   1:L PR[91] 10mm/sec CNT100;
   1:  PR[GP1:91,1] = PR[GP1:90,1] + -17.777;
   1:  PR[GP1:91,2] = PR[GP1:90,2] + -17.049;
   1:L PR[91] 10mm/sec CNT100;
   1:  PR[GP1:91,1] = PR[GP1:90,1] + -17.068;
   1:  PR[GP1:91,2] = PR[GP1:90,2] + -16.935;
   1:L PR[91] 10mm/sec CNT100;
   1:  PR[GP1:91,1] = PR[GP1:90,1] + -14.386;
   1:  PR[GP1:91,2] = PR[GP1:90,2] + -16.296;
   1:L PR[91] 10mm/sec CNT100;
   1:  PR[GP1:91,1] = PR[GP1:90,1] + -13.899;
   1:  PR[GP1:91,2] = PR[GP1:90,2] + -16.133;
   1:L PR[91] 10mm/sec CNT100;
   1:  PR[GP1:91,1] = PR[GP1:90,1] + -11.116;
   1:  PR[GP1:91,2] = PR[GP1:90,2] + -14.804;
   1:L PR[91] 10mm/sec CNT100;
   1:  PR[GP1:91,1] = PR[GP1:90,1] + -10.848;
   1:  PR[GP1:91,2] = PR[GP1:90,2] + -14.661;
   1:L PR[91] 10mm/sec CNT100;
   1:  PR[GP1:91,1] = PR[GP1:90,1] + -8.058;
   1:  PR[GP1:91,2] = PR[GP1:90,2] + -12.514;
   1:L PR[91] 10mm/sec CNT100;
   1:  PR[GP1:91,1] = PR[GP1:90,1] + -7.983;
   1:  PR[GP1:91,2] = PR[GP1:90,2] + -12.434;
   1:L PR[91] 10mm/sec CNT100;
   1:  PR[GP1:91,1] = PR[GP1:90,1] + -5.754;
   1:  PR[GP1:91,2] = PR[GP1:90,2] + -9.796;
   1:L PR[91] 10mm/sec CNT100;
   1:  PR[GP1:91,1] = PR[GP1:90,1] + -4.074;
   1:  PR[GP1:91,2] = PR[GP1:90,2] + -6.675;
   1:L PR[91] 10mm/sec CNT100;
   1:  PR[GP1:91,1] = PR[GP1:90,1] + -3.054;
   1:  PR[GP1:91,2] = PR[GP1:90,2] + -3.139;
   1:L PR[91] 10mm/sec CNT100;
   1:  PR[GP1:91,1] = PR[GP1:90,1] + -2.957;
   1:  PR[GP1:91,2] = PR[GP1:90,2] + -2.843;
   1:L PR[91] 10mm/sec CNT100;
   1:  PR[GP1:91,1] = PR[GP1:90,1] + -2.891;
   1:  PR[GP1:91,2] = PR[GP1:90,2] + -2.753;
   1:L PR[91] 10mm/sec CNT100;
   1:  PR[GP1:91,1] = PR[GP1:90,1] + -2.846;
   1:  PR[GP1:91,2] = PR[GP1:90,2] + -2.649;
   1:L PR[91] 10mm/sec CNT100;
   1:  PR[GP1:91,1] = PR[GP1:90,1] + -2.751;
   1:  PR[GP1:91,2] = PR[GP1:90,2] + -2.377;
   1:L PR[91] 10mm/sec CNT100;
   1:  PR[GP1:91,1] = PR[GP1:90,1] + -2.564;
   1:  PR[GP1:91,2] = PR[GP1:90,2] + -2.018;
   1:L PR[91] 10mm/sec CNT100;
   1:  PR[GP1:91,1] = PR[GP1:90,1] + -2.286;
   1:  PR[GP1:91,2] = PR[GP1:90,2] + -1.644;
   1:L PR[91] 10mm/sec CNT100;
   1:  PR[GP1:91,1] = PR[GP1:90,1] + -1.981;
   1:  PR[GP1:91,2] = PR[GP1:90,2] + -1.337;
   1:L PR[91] 10mm/sec CNT100;
   1:  PR[GP1:91,1] = PR[GP1:90,1] + -1.497;
   1:  PR[GP1:91,2] = PR[GP1:90,2] + -1.028;
   1:L PR[91] 10mm/sec CNT100;
   1:  PR[GP1:91,1] = PR[GP1:90,1] + -1.290;
   1:  PR[GP1:91,2] = PR[GP1:90,2] + -0.917;
   1:L PR[91] 10mm/sec CNT100;
   1:  PR[GP1:91,1] = PR[GP1:90,1] + -0.204;
   1:  PR[GP1:91,2] = PR[GP1:90,2] + -0.687;
   1:L PR[91] 10mm/sec CNT100;
   1:  PR[GP1:91,1] = PR[GP1:90,1] + 0.891;
   1:  PR[GP1:91,2] = PR[GP1:90,2] + -0.965;
   1:L PR[91] 10mm/sec CNT100;
   1:  PR[GP1:91,1] = PR[GP1:90,1] + 1.190;
   1:  PR[GP1:91,2] = PR[GP1:90,2] + -1.125;
   1:L PR[91] 10mm/sec CNT100;
   1:  PR[GP1:91,1] = PR[GP1:90,1] + 1.414;
   1:  PR[GP1:91,2] = PR[GP1:90,2] + -1.278;
   1:L PR[91] 10mm/sec CNT100;
   1:  PR[GP1:91,1] = PR[GP1:90,1] + 2.090;
   1:  PR[GP1:91,2] = PR[GP1:90,2] + -1.951;
   1:L PR[91] 10mm/sec CNT100;
   1:  PR[GP1:91,1] = PR[GP1:90,1] + 2.234;
   1:  PR[GP1:91,2] = PR[GP1:90,2] + -2.141;
   1:L PR[91] 10mm/sec CNT100;
   1:  PR[GP1:91,1] = PR[GP1:90,1] + 2.617;
   1:  PR[GP1:91,2] = PR[GP1:90,2] + -3.082;
   1:L PR[91] 10mm/sec CNT100;
   1:  PR[GP1:91,1] = PR[GP1:90,1] + 3.318;
   1:  PR[GP1:91,2] = PR[GP1:90,2] + -5.804;
   1:L PR[91] 10mm/sec CNT100;
   1:  PR[GP1:91,1] = PR[GP1:90,1] + 4.418;
   1:  PR[GP1:91,2] = PR[GP1:90,2] + -8.231;
   1:L PR[91] 10mm/sec CNT100;
   1:  PR[GP1:91,1] = PR[GP1:90,1] + 5.923;
   1:  PR[GP1:91,2] = PR[GP1:90,2] + -10.467;
   1:L PR[91] 10mm/sec CNT100;
   1:  PR[GP1:91,1] = PR[GP1:90,1] + 7.757;
   1:  PR[GP1:91,2] = PR[GP1:90,2] + -12.452;
   1:L PR[91] 10mm/sec CNT100;
   1:  PR[GP1:91,1] = PR[GP1:90,1] + 9.893;
   1:  PR[GP1:91,2] = PR[GP1:90,2] + -14.128;
   1:L PR[91] 10mm/sec CNT100;
   1:  PR[GP1:91,1] = PR[GP1:90,1] + 12.262;
   1:  PR[GP1:91,2] = PR[GP1:90,2] + -15.460;
   1:L PR[91] 10mm/sec CNT100;
   1:  PR[GP1:91,1] = PR[GP1:90,1] + 14.756;
   1:  PR[GP1:91,2] = PR[GP1:90,2] + -16.425;
   1:L PR[91] 10mm/sec CNT100;
   1:  PR[GP1:91,1] = PR[GP1:90,1] + 17.367;
   1:  PR[GP1:91,2] = PR[GP1:90,2] + -16.996;
   1:L PR[91] 10mm/sec CNT100;
   1:  PR[GP1:91,1] = PR[GP1:90,1] + 20.036;
   1:  PR[GP1:91,2] = PR[GP1:90,2] + -17.161;
   1:L PR[91] 10mm/sec CNT100;
   1:  PR[GP1:91,1] = PR[GP1:90,1] + 22.699;
   1:  PR[GP1:91,2] = PR[GP1:90,2] + -16.917;
   1:L PR[91] 10mm/sec CNT100;
   1:  PR[GP1:91,1] = PR[GP1:90,1] + 25.303;
   1:  PR[GP1:91,2] = PR[GP1:90,2] + -16.264;
   1:L PR[91] 10mm/sec CNT100;
   1:  PR[GP1:91,1] = PR[GP1:90,1] + 27.687;
   1:  PR[GP1:91,2] = PR[GP1:90,2] + -15.253;
   1:L PR[91] 10mm/sec CNT100;
   1:  PR[GP1:91,1] = PR[GP1:90,1] + 29.800;
   1:  PR[GP1:91,2] = PR[GP1:90,2] + -13.948;
   1:L PR[91] 10mm/sec CNT100;
   1:  PR[GP1:91,1] = PR[GP1:90,1] + 30.069;
   1:  PR[GP1:91,2] = PR[GP1:90,2] + -13.749;
   1:L PR[91] 10mm/sec CNT100;
   1:  PR[GP1:91,1] = PR[GP1:90,1] + 31.620;
   1:  PR[GP1:91,2] = PR[GP1:90,2] + -12.411;
   1:L PR[91] 10mm/sec CNT100;
   1:  PR[GP1:91,1] = PR[GP1:90,1] + 31.946;
   1:  PR[GP1:91,2] = PR[GP1:90,2] + -12.109;
   1:L PR[91] 10mm/sec CNT100;
   1:  PR[GP1:91,1] = PR[GP1:90,1] + 33.516;
   1:  PR[GP1:91,2] = PR[GP1:90,2] + -10.262;
   1:L PR[91] 10mm/sec CNT100;
   1:  PR[GP1:91,1] = PR[GP1:90,1] + 33.815;
   1:  PR[GP1:91,2] = PR[GP1:90,2] + -9.828;
   1:L PR[91] 10mm/sec CNT100;
   1:  PR[GP1:91,1] = PR[GP1:90,1] + 34.762;
   1:  PR[GP1:91,2] = PR[GP1:90,2] + -8.269;
   1:L PR[91] 10mm/sec CNT100;
   1:  PR[GP1:91,1] = PR[GP1:90,1] + 35.043;
   1:  PR[GP1:91,2] = PR[GP1:90,2] + -7.748;
   1:L PR[91] 10mm/sec CNT100;
   1:  PR[GP1:91,1] = PR[GP1:90,1] + 35.944;
   1:  PR[GP1:91,2] = PR[GP1:90,2] + -5.545;
   1:L PR[91] 10mm/sec CNT100;
   1:  PR[GP1:91,1] = PR[GP1:90,1] + 36.117;
   1:  PR[GP1:91,2] = PR[GP1:90,2] + -4.929;
   1:L PR[91] 10mm/sec CNT100;
   1:  PR[GP1:91,1] = PR[GP1:90,1] + 36.509;
   1:  PR[GP1:91,2] = PR[GP1:90,2] + -3.281;
   1:L PR[91] 10mm/sec CNT100;
   1:  PR[GP1:91,1] = PR[GP1:90,1] + 36.618;
   1:  PR[GP1:91,2] = PR[GP1:90,2] + -2.625;
   1:L PR[91] 10mm/sec CNT100;
   1:  PR[GP1:91,1] = PR[GP1:90,1] + 36.657;
   1:  PR[GP1:91,2] = PR[GP1:90,2] + -1.925;
   1:L PR[91] 10mm/sec CNT100;
   1:  PR[GP1:91,1] = PR[GP1:90,1] + 36.816;
   1:  PR[GP1:91,2] = PR[GP1:90,2] + -0.277;
   1:L PR[91] 10mm/sec CNT100;
   1:  PR[GP1:91,1] = PR[GP1:90,1] + 36.466;
   1:  PR[GP1:91,2] = PR[GP1:90,2] + 3.030;
   1:L PR[91] 10mm/sec CNT100;
   1:  PR[GP1:91,1] = PR[GP1:90,1] + 35.808;
   1:  PR[GP1:91,2] = PR[GP1:90,2] + 5.173;
   1:L PR[91] 10mm/sec CNT100;
   1:  PR[GP1:91,1] = PR[GP1:90,1] + 35.611;
   1:  PR[GP1:91,2] = PR[GP1:90,2] + 5.902;
   1:L PR[91] 10mm/sec CNT100;
   1:  PR[GP1:91,1] = PR[GP1:90,1] + 35.499;
   1:  PR[GP1:91,2] = PR[GP1:90,2] + 6.196;
   1:L PR[91] 10mm/sec CNT100;
   1:  PR[GP1:91,1] = PR[GP1:90,1] + 33.908;
   1:  PR[GP1:91,2] = PR[GP1:90,2] + 9.143;
   1:L PR[91] 10mm/sec CNT100;
   1:  PR[GP1:91,1] = PR[GP1:90,1] + 32.344;
   1:  PR[GP1:91,2] = PR[GP1:90,2] + 11.025;
   1:L PR[91] 10mm/sec CNT100;
   1:  PR[GP1:91,1] = PR[GP1:90,1] + 32.162;
   1:  PR[GP1:91,2] = PR[GP1:90,2] + 11.277;
   1:L PR[91] 10mm/sec CNT100;
   1:  PR[GP1:91,1] = PR[GP1:90,1] + 31.790;
   1:  PR[GP1:91,2] = PR[GP1:90,2] + 11.697;
   1:L PR[91] 10mm/sec CNT100;
   1:  PR[GP1:91,1] = PR[GP1:90,1] + 29.195;
   1:  PR[GP1:91,2] = PR[GP1:90,2] + 13.796;
   1:L PR[91] 10mm/sec CNT100;
   1:  PR[GP1:91,1] = PR[GP1:90,1] + 26.248;
   1:  PR[GP1:91,2] = PR[GP1:90,2] + 15.339;
   1:L PR[91] 10mm/sec CNT100;
   1:  PR[GP1:91,1] = PR[GP1:90,1] + 23.089;
   1:  PR[GP1:91,2] = PR[GP1:90,2] + 16.266;
   1:L PR[91] 10mm/sec CNT100;
   1:  PR[GP1:91,1] = PR[GP1:90,1] + 19.713;
   1:  PR[GP1:91,2] = PR[GP1:90,2] + 16.557;
   1:L PR[91] 10mm/sec CNT100;
   1:  PR[GP1:91,1] = PR[GP1:90,1] + 16.351;
   1:  PR[GP1:91,2] = PR[GP1:90,2] + 16.182;
   1:L PR[91] 10mm/sec CNT100;
   1:  PR[GP1:91,1] = PR[GP1:90,1] + 13.131;
   1:  PR[GP1:91,2] = PR[GP1:90,2] + 15.163;
   1:L PR[91] 10mm/sec CNT100;
   1:  PR[GP1:91,1] = PR[GP1:90,1] + 10.178;
   1:  PR[GP1:91,2] = PR[GP1:90,2] + 13.541;
   1:L PR[91] 10mm/sec CNT100;
   1:  PR[GP1:91,1] = PR[GP1:90,1] + 7.542;
   1:  PR[GP1:91,2] = PR[GP1:90,2] + 11.371;
   1:L PR[91] 10mm/sec CNT100;
   1:  PR[GP1:91,1] = PR[GP1:90,1] + 5.385;
   1:  PR[GP1:91,2] = PR[GP1:90,2] + 8.744;
   1:L PR[91] 10mm/sec CNT100;
   1:  PR[GP1:91,1] = PR[GP1:90,1] + 3.746;
   1:  PR[GP1:91,2] = PR[GP1:90,2] + 5.756;
   1:L PR[91] 10mm/sec CNT100;
   1:  PR[GP1:91,1] = PR[GP1:90,1] + 2.740;
   1:  PR[GP1:91,2] = PR[GP1:90,2] + 2.534;
   1:L PR[91] 10mm/sec CNT100;
   1:  PR[GP1:91,1] = PR[GP1:90,1] + 2.273;
   1:  PR[GP1:91,2] = PR[GP1:90,2] + 1.475;
   1:L PR[91] 10mm/sec CNT100;
   1:  PR[GP1:91,1] = PR[GP1:90,1] + 1.462;
   1:  PR[GP1:91,2] = PR[GP1:90,2] + 0.697;
   1:L PR[91] 10mm/sec CNT100;
   1:  PR[GP1:91,1] = PR[GP1:90,1] + 1.135;
   1:  PR[GP1:91,2] = PR[GP1:90,2] + 0.502;
   1:L PR[91] 10mm/sec CNT100;
   1:  PR[GP1:91,1] = PR[GP1:90,1] + 0.670;
   1:  PR[GP1:91,2] = PR[GP1:90,2] + 0.285;
   1:L PR[91] 10mm/sec CNT100;
   1:  PR[GP1:91,1] = PR[GP1:90,1] + -0.451;
   1:  PR[GP1:91,2] = PR[GP1:90,2] + 0.136;
   1:L PR[91] 10mm/sec CNT100;
   1:  PR[GP1:91,1] = PR[GP1:90,1] + -1.415;
   1:  PR[GP1:91,2] = PR[GP1:90,2] + 0.419;
   1:L PR[91] 10mm/sec CNT100;
   1:  PR[GP1:91,1] = PR[GP1:90,1] + -1.565;
   1:  PR[GP1:91,2] = PR[GP1:90,2] + 0.501;
   1:L PR[91] 10mm/sec CNT100;
   1:  PR[GP1:91,1] = PR[GP1:90,1] + -1.924;
   1:  PR[GP1:91,2] = PR[GP1:90,2] + 0.759;
   1:L PR[91] 10mm/sec CNT100;
   1:  PR[GP1:91,1] = PR[GP1:90,1] + -2.230;
   1:  PR[GP1:91,2] = PR[GP1:90,2] + 1.037;
   1:L PR[91] 10mm/sec CNT100;
   1:  PR[GP1:91,1] = PR[GP1:90,1] + -2.571;
   1:  PR[GP1:91,2] = PR[GP1:90,2] + 1.459;
   1:L PR[91] 10mm/sec CNT100;
   1:  PR[GP1:91,1] = PR[GP1:90,1] + -2.686;
   1:  PR[GP1:91,2] = PR[GP1:90,2] + 1.725;
   1:L PR[91] 10mm/sec CNT100;
   1:  PR[GP1:91,1] = PR[GP1:90,1] + -2.840;
   1:  PR[GP1:91,2] = PR[GP1:90,2] + 2.011;
   1:L PR[91] 10mm/sec CNT100;
   1:  PR[GP1:91,1] = PR[GP1:90,1] + -2.897;
   1:  PR[GP1:91,2] = PR[GP1:90,2] + 2.157;
   1:L PR[91] 10mm/sec CNT100;
   1:  PR[GP1:91,1] = PR[GP1:90,1] + -2.963;
   1:  PR[GP1:91,2] = PR[GP1:90,2] + 2.160;
   1:L PR[91] 10mm/sec CNT100;
   1:  PR[GP1:91,1] = PR[GP1:90,1] + -4.071;
   1:  PR[GP1:91,2] = PR[GP1:90,2] + 6.022;
   1:L PR[91] 10mm/sec CNT100;
   1:  PR[GP1:91,1] = PR[GP1:90,1] + -4.185;
   1:  PR[GP1:91,2] = PR[GP1:90,2] + 6.274;
   1:L PR[91] 10mm/sec CNT100;
   1:  PR[GP1:91,1] = PR[GP1:90,1] + -5.644;
   1:  PR[GP1:91,2] = PR[GP1:90,2] + 8.982;
   1:L PR[91] 10mm/sec CNT100;
   1:  PR[GP1:91,1] = PR[GP1:90,1] + -5.914;
   1:  PR[GP1:91,2] = PR[GP1:90,2] + 9.386;
   1:L PR[91] 10mm/sec CNT100;
   1:  PR[GP1:91,1] = PR[GP1:90,1] + -7.700;
   1:  PR[GP1:91,2] = PR[GP1:90,2] + 11.479;
   1:L PR[91] 10mm/sec CNT100;
   1:  PR[GP1:91,1] = PR[GP1:90,1] + -8.173;
   1:  PR[GP1:91,2] = PR[GP1:90,2] + 11.985;
   1:L PR[91] 10mm/sec CNT100;
   1:  PR[GP1:91,1] = PR[GP1:90,1] + -10.830;
   1:  PR[GP1:91,2] = PR[GP1:90,2] + 14.014;
   1:L PR[91] 10mm/sec CNT100;
   1:  PR[GP1:91,1] = PR[GP1:90,1] + -11.609;
   1:  PR[GP1:91,2] = PR[GP1:90,2] + 14.428;
   1:L PR[91] 10mm/sec CNT100;
   1:  PR[GP1:91,1] = PR[GP1:90,1] + -13.732;
   1:  PR[GP1:91,2] = PR[GP1:90,2] + 15.431;
   1:L PR[91] 10mm/sec CNT100;
   1:  PR[GP1:91,1] = PR[GP1:90,1] + -14.726;
   1:  PR[GP1:91,2] = PR[GP1:90,2] + 15.765;
   1:L PR[91] 10mm/sec CNT100;
   1:  PR[GP1:91,1] = PR[GP1:90,1] + -16.776;
   1:  PR[GP1:91,2] = PR[GP1:90,2] + 16.244;
   1:L PR[91] 10mm/sec CNT100;
   1:  PR[GP1:91,1] = PR[GP1:90,1] + -17.943;
   1:  PR[GP1:91,2] = PR[GP1:90,2] + 16.432;
   1:L PR[91] 10mm/sec CNT100;
   1:  PR[GP1:91,1] = PR[GP1:90,1] + -19.155;
   1:  PR[GP1:91,2] = PR[GP1:90,2] + 16.425;
   1:L PR[91] 10mm/sec CNT100;
   1:  PR[GP1:91,1] = PR[GP1:90,1] + -21.180;
   1:  PR[GP1:91,2] = PR[GP1:90,2] + 16.457;
   1:L PR[91] 10mm/sec CNT100;
   1:  PR[GP1:91,1] = PR[GP1:90,1] + -22.467;
   1:  PR[GP1:91,2] = PR[GP1:90,2] + 16.236;
   1:L PR[91] 10mm/sec CNT100;
   1:  PR[GP1:91,1] = PR[GP1:90,1] + -24.282;
   1:  PR[GP1:91,2] = PR[GP1:90,2] + 15.879;
   1:L PR[91] 10mm/sec CNT100;
   1:  PR[GP1:91,1] = PR[GP1:90,1] + -25.602;
   1:  PR[GP1:91,2] = PR[GP1:90,2] + 15.419;
   1:L PR[91] 10mm/sec CNT100;
   1:  PR[GP1:91,1] = PR[GP1:90,1] + -27.180;
   1:  PR[GP1:91,2] = PR[GP1:90,2] + 14.741;
   1:L PR[91] 10mm/sec CNT100;
   1:  PR[GP1:91,1] = PR[GP1:90,1] + -28.470;
   1:  PR[GP1:91,2] = PR[GP1:90,2] + 14.037;
   1:L PR[91] 10mm/sec CNT100;
   1:  PR[GP1:91,1] = PR[GP1:90,1] + -29.792;
   1:  PR[GP1:91,2] = PR[GP1:90,2] + 13.097;
   1:L PR[91] 10mm/sec CNT100;
   1:  PR[GP1:91,1] = PR[GP1:90,1] + -30.990;
   1:  PR[GP1:91,2] = PR[GP1:90,2] + 12.159;
   1:L PR[91] 10mm/sec CNT100;
   1:  PR[GP1:91,1] = PR[GP1:90,1] + -33.104;
   1:  PR[GP1:91,2] = PR[GP1:90,2] + 9.848;
   1:L PR[91] 10mm/sec CNT100;
   1:  PR[GP1:91,1] = PR[GP1:90,1] + -33.952;
   1:  PR[GP1:91,2] = PR[GP1:90,2] + 8.545;
   1:L PR[91] 10mm/sec CNT100;
   1:  PR[GP1:91,1] = PR[GP1:90,1] + -34.734;
   1:  PR[GP1:91,2] = PR[GP1:90,2] + 7.207;
   1:L PR[91] 10mm/sec CNT100;
   1:  PR[GP1:91,1] = PR[GP1:90,1] + -35.363;
   1:  PR[GP1:91,2] = PR[GP1:90,2] + 5.766;
   1:L PR[91] 10mm/sec CNT100;
   1:  PR[GP1:91,1] = PR[GP1:90,1] + -35.844;
   1:  PR[GP1:91,2] = PR[GP1:90,2] + 4.309;
   1:L PR[91] 10mm/sec CNT100;
   1:  PR[GP1:91,1] = PR[GP1:90,1] + -36.227;
   1:  PR[GP1:91,2] = PR[GP1:90,2] + 2.791;
   1:L PR[91] 10mm/sec CNT100;
   1:  PR[GP1:91,1] = PR[GP1:90,1] + -36.358;
   1:  PR[GP1:91,2] = PR[GP1:90,2] + 1.200;
   1:L PR[91] 10mm/sec CNT100;
   1:  PR[GP1:91,1] = PR[GP1:90,1] + -36.519;
   1:  PR[GP1:91,2] = PR[GP1:90,2] + -0.326;
   1:L PR[91] 10mm/sec CNT100;
   1:  PR[GP1:91,1] = PR[GP1:90,1] + -36.391;
   1:  PR[GP1:91,2] = PR[GP1:90,2] + -1.877;
   1:L PR[91] 10mm/sec CNT100;
   1:  PR[GP1:91,1] = PR[GP1:90,1] + -36.222;
   1:  PR[GP1:91,2] = PR[GP1:90,2] + -3.434;
   1:L PR[91] 10mm/sec CNT100;
   1:  PR[GP1:91,1] = PR[GP1:90,1] + -35.849;
   1:  PR[GP1:91,2] = PR[GP1:90,2] + -4.915;
   1:L PR[91] 10mm/sec CNT100;
   1:  PR[GP1:91,1] = PR[GP1:90,1] + -35.341;
   1:  PR[GP1:91,2] = PR[GP1:90,2] + -6.456;
   1:L PR[91] 10mm/sec CNT100;
   1:  PR[GP1:91,1] = PR[GP1:90,1] + -34.749;
   1:  PR[GP1:91,2] = PR[GP1:90,2] + -7.810;
   1:L PR[91] 10mm/sec CNT100;
   1:  PR[GP1:91,1] = PR[GP1:90,1] + -33.879;
   1:  PR[GP1:91,2] = PR[GP1:90,2] + -9.291;
   1:L PR[91] 10mm/sec CNT100;
   1:  PR[GP1:91,1] = PR[GP1:90,1] + -33.110;
   1:  PR[GP1:91,2] = PR[GP1:90,2] + -10.473;
   1:L PR[91] 10mm/sec CNT100;
   1:  PR[GP1:91,1] = PR[GP1:90,1] + -30.957;
   1:  PR[GP1:91,2] = PR[GP1:90,2] + -12.821;
   1:L PR[91] 10mm/sec CNT100;
   1:  PR[GP1:91,1] = PR[GP1:90,1] + -29.919;
   1:  PR[GP1:91,2] = PR[GP1:90,2] + -13.635;
   1:L PR[91] 10mm/sec CNT100;
   1:  PR[GP1:91,1] = PR[GP1:90,1] + -28.357;
   1:  PR[GP1:91,2] = PR[GP1:90,2] + -14.738;
   1:L PR[91] 10mm/sec CNT100;
   1:  PR[GP1:91,1] = PR[GP1:90,1] + -27.298;
   1:  PR[GP1:91,2] = PR[GP1:90,2] + -15.316;
   1:L PR[91] 10mm/sec CNT100;
   1:  PR[GP1:91,1] = PR[GP1:90,1] + -25.359;
   1:  PR[GP1:91,2] = PR[GP1:90,2] + -16.142;
   1:L PR[91] 10mm/sec CNT100;
   1:  PR[GP1:91,1] = PR[GP1:90,1] + -24.356;
   1:  PR[GP1:91,2] = PR[GP1:90,2] + -16.491;
   1:L PR[91] 10mm/sec CNT100;
   1:  PR[GP1:91,1] = PR[GP1:90,1] + -23.976;
   1:  PR[GP1:91,2] = PR[GP1:90,2] + -16.549;
   1:  PR[GP1:91,3] = PR[GP1:90,3] + 8.800;
   1:L PR[91] 10mm/sec CNT100;
   1:  PR[GP1:91,1] = PR[GP1:90,1] + -21.062;
   1:  PR[GP1:91,2] = PR[GP1:90,2] + -17.118;
   1:L PR[91] 10mm/sec CNT100;
   1:  PR[GP1:91,1] = PR[GP1:90,1] + -20.821;
   1:  PR[GP1:91,2] = PR[GP1:90,2] + -17.119;
   1:L PR[91] 10mm/sec CNT100;
   1:  PR[GP1:91,1] = PR[GP1:90,1] + -17.518;
   1:  PR[GP1:91,2] = PR[GP1:90,2] + -17.049;
   1:L PR[91] 10mm/sec CNT100;
   1:  PR[GP1:91,1] = PR[GP1:90,1] + -14.070;
   1:  PR[GP1:91,2] = PR[GP1:90,2] + -16.265;
   1:L PR[91] 10mm/sec CNT100;
   1:  PR[GP1:91,1] = PR[GP1:90,1] + -13.874;
   1:  PR[GP1:91,2] = PR[GP1:90,2] + -16.195;
   1:L PR[91] 10mm/sec CNT100;
   1:  PR[GP1:91,1] = PR[GP1:90,1] + -10.954;
   1:  PR[GP1:91,2] = PR[GP1:90,2] + -14.845;
   1:L PR[91] 10mm/sec CNT100;
   1:  PR[GP1:91,1] = PR[GP1:90,1] + -10.479;
   1:  PR[GP1:91,2] = PR[GP1:90,2] + -14.558;
   1:L PR[91] 10mm/sec CNT100;
   1:  PR[GP1:91,1] = PR[GP1:90,1] + -8.213;
   1:  PR[GP1:91,2] = PR[GP1:90,2] + -12.849;
   1:L PR[91] 10mm/sec CNT100;
   1:  PR[GP1:91,1] = PR[GP1:90,1] + -7.582;
   1:  PR[GP1:91,2] = PR[GP1:90,2] + -12.265;
   1:L PR[91] 10mm/sec CNT100;
   1:  PR[GP1:91,1] = PR[GP1:90,1] + -5.938;
   1:  PR[GP1:91,2] = PR[GP1:90,2] + -10.352;
   1:L PR[91] 10mm/sec CNT100;
   1:  PR[GP1:91,1] = PR[GP1:90,1] + -5.301;
   1:  PR[GP1:91,2] = PR[GP1:90,2] + -9.461;
   1:L PR[91] 10mm/sec CNT100;
   1:  PR[GP1:91,1] = PR[GP1:90,1] + -4.202;
   1:  PR[GP1:91,2] = PR[GP1:90,2] + -7.423;
   1:L PR[91] 10mm/sec CNT100;
   1:  PR[GP1:91,1] = PR[GP1:90,1] + -3.704;
   1:  PR[GP1:91,2] = PR[GP1:90,2] + -6.304;
   1:L PR[91] 10mm/sec CNT100;
   1:  PR[GP1:91,1] = PR[GP1:90,1] + -3.091;
   1:  PR[GP1:91,2] = PR[GP1:90,2] + -4.168;
   1:L PR[91] 10mm/sec CNT100;
   1:  PR[GP1:91,1] = PR[GP1:90,1] + -2.973;
   1:  PR[GP1:91,2] = PR[GP1:90,2] + -3.559;
   1:L PR[91] 10mm/sec CNT100;
   1:  PR[GP1:91,1] = PR[GP1:90,1] + -2.742;
   1:  PR[GP1:91,2] = PR[GP1:90,2] + -2.960;
   1:L PR[91] 10mm/sec CNT100;
   1:  PR[GP1:91,1] = PR[GP1:90,1] + -2.498;
   1:  PR[GP1:91,2] = PR[GP1:90,2] + -2.246;
   1:L PR[91] 10mm/sec CNT100;
   1:  PR[GP1:91,1] = PR[GP1:90,1] + -2.348;
   1:  PR[GP1:91,2] = PR[GP1:90,2] + -2.123;
   1:L PR[91] 10mm/sec CNT100;
   1:  PR[GP1:91,1] = PR[GP1:90,1] + -2.298;
   1:  PR[GP1:91,2] = PR[GP1:90,2] + -2.054;
   1:L PR[91] 10mm/sec CNT100;
   1:  PR[GP1:91,1] = PR[GP1:90,1] + -1.650;
   1:  PR[GP1:91,2] = PR[GP1:90,2] + -1.402;
   1:L PR[91] 10mm/sec CNT100;
   1:  PR[GP1:91,1] = PR[GP1:90,1] + -1.350;
   1:  PR[GP1:91,2] = PR[GP1:90,2] + -1.336;
   1:L PR[91] 10mm/sec CNT100;
   1:  PR[GP1:91,1] = PR[GP1:90,1] + -0.557;
   1:  PR[GP1:91,2] = PR[GP1:90,2] + -1.032;
   1:L PR[91] 10mm/sec CNT100;
   1:  PR[GP1:91,1] = PR[GP1:90,1] + 0.704;
   1:  PR[GP1:91,2] = PR[GP1:90,2] + -1.259;
   1:L PR[91] 10mm/sec CNT100;
   1:  PR[GP1:91,1] = PR[GP1:90,1] + 1.056;
   1:  PR[GP1:91,2] = PR[GP1:90,2] + -1.522;
   1:L PR[91] 10mm/sec CNT100;
   1:  PR[GP1:91,1] = PR[GP1:90,1] + 1.863;
   1:  PR[GP1:91,2] = PR[GP1:90,2] + -2.364;
   1:L PR[91] 10mm/sec CNT100;
   1:  PR[GP1:91,1] = PR[GP1:90,1] + 2.057;
   1:  PR[GP1:91,2] = PR[GP1:90,2] + -2.848;
   1:L PR[91] 10mm/sec CNT100;
   1:  PR[GP1:91,1] = PR[GP1:90,1] + 2.821;
   1:  PR[GP1:91,2] = PR[GP1:90,2] + -5.845;
   1:L PR[91] 10mm/sec CNT100;
   1:  PR[GP1:91,1] = PR[GP1:90,1] + 3.917;
   1:  PR[GP1:91,2] = PR[GP1:90,2] + -8.286;
   1:L PR[91] 10mm/sec CNT100;
   1:  PR[GP1:91,1] = PR[GP1:90,1] + 5.426;
   1:  PR[GP1:91,2] = PR[GP1:90,2] + -10.530;
   1:L PR[91] 10mm/sec CNT100;
   1:  PR[GP1:91,1] = PR[GP1:90,1] + 7.308;
   1:  PR[GP1:91,2] = PR[GP1:90,2] + -12.517;
   1:L PR[91] 10mm/sec CNT100;
   1:  PR[GP1:91,1] = PR[GP1:90,1] + 9.508;
   1:  PR[GP1:91,2] = PR[GP1:90,2] + -14.197;
   1:L PR[91] 10mm/sec CNT100;
   1:  PR[GP1:91,1] = PR[GP1:90,1] + 11.906;
   1:  PR[GP1:91,2] = PR[GP1:90,2] + -15.534;
   1:L PR[91] 10mm/sec CNT100;
   1:  PR[GP1:91,1] = PR[GP1:90,1] + 14.486;
   1:  PR[GP1:91,2] = PR[GP1:90,2] + -16.488;
   1:L PR[91] 10mm/sec CNT100;
   1:  PR[GP1:91,1] = PR[GP1:90,1] + 17.160;
   1:  PR[GP1:91,2] = PR[GP1:90,2] + -17.049;
   1:L PR[91] 10mm/sec CNT100;
   1:  PR[GP1:91,1] = PR[GP1:90,1] + 19.836;
   1:  PR[GP1:91,2] = PR[GP1:90,2] + -17.211;
   1:L PR[91] 10mm/sec CNT100;
   1:  PR[GP1:91,1] = PR[GP1:90,1] + 22.503;
   1:  PR[GP1:91,2] = PR[GP1:90,2] + -16.963;
   1:L PR[91] 10mm/sec CNT100;
   1:  PR[GP1:91,1] = PR[GP1:90,1] + 25.099;
   1:  PR[GP1:91,2] = PR[GP1:90,2] + -16.312;
   1:L PR[91] 10mm/sec CNT100;
   1:  PR[GP1:91,1] = PR[GP1:90,1] + 27.562;
   1:  PR[GP1:91,2] = PR[GP1:90,2] + -15.274;
   1:L PR[91] 10mm/sec CNT100;
   1:  PR[GP1:91,1] = PR[GP1:90,1] + 29.832;
   1:  PR[GP1:91,2] = PR[GP1:90,2] + -13.874;
   1:L PR[91] 10mm/sec CNT100;
   1:  PR[GP1:91,1] = PR[GP1:90,1] + 31.852;
   1:  PR[GP1:91,2] = PR[GP1:90,2] + -12.148;
   1:L PR[91] 10mm/sec CNT100;
   1:  PR[GP1:91,1] = PR[GP1:90,1] + 33.526;
   1:  PR[GP1:91,2] = PR[GP1:90,2] + -10.169;
   1:L PR[91] 10mm/sec CNT100;
   1:  PR[GP1:91,1] = PR[GP1:90,1] + 34.933;
   1:  PR[GP1:91,2] = PR[GP1:90,2] + -7.847;
   1:L PR[91] 10mm/sec CNT100;
   1:  PR[GP1:91,1] = PR[GP1:90,1] + 35.895;
   1:  PR[GP1:91,2] = PR[GP1:90,2] + -5.500;
   1:L PR[91] 10mm/sec CNT100;
   1:  PR[GP1:91,1] = PR[GP1:90,1] + 36.489;
   1:  PR[GP1:91,2] = PR[GP1:90,2] + -3.049;
   1:L PR[91] 10mm/sec CNT100;
   1:  PR[GP1:91,1] = PR[GP1:90,1] + 36.529;
   1:  PR[GP1:91,2] = PR[GP1:90,2] + -2.807;
   1:L PR[91] 10mm/sec CNT100;
   1:  PR[GP1:91,1] = PR[GP1:90,1] + 36.544;
   1:  PR[GP1:91,2] = PR[GP1:90,2] + -2.524;
   1:L PR[91] 10mm/sec CNT100;
   1:  PR[GP1:91,1] = PR[GP1:90,1] + 36.759;
   1:  PR[GP1:91,2] = PR[GP1:90,2] + -0.283;
   1:L PR[91] 10mm/sec CNT100;
   1:  PR[GP1:91,1] = PR[GP1:90,1] + 36.403;
   1:  PR[GP1:91,2] = PR[GP1:90,2] + 3.024;
   1:L PR[91] 10mm/sec CNT100;
   1:  PR[GP1:91,1] = PR[GP1:90,1] + 35.425;
   1:  PR[GP1:91,2] = PR[GP1:90,2] + 6.209;
   1:L PR[91] 10mm/sec CNT100;
   1:  PR[GP1:91,1] = PR[GP1:90,1] + 33.843;
   1:  PR[GP1:91,2] = PR[GP1:90,2] + 9.138;
   1:L PR[91] 10mm/sec CNT100;
   1:  PR[GP1:91,1] = PR[GP1:90,1] + 31.716;
   1:  PR[GP1:91,2] = PR[GP1:90,2] + 11.698;
   1:L PR[91] 10mm/sec CNT100;
   1:  PR[GP1:91,1] = PR[GP1:90,1] + 30.650;
   1:  PR[GP1:91,2] = PR[GP1:90,2] + 12.561;
   1:L PR[91] 10mm/sec CNT100;
   1:  PR[GP1:91,1] = PR[GP1:90,1] + 29.111;
   1:  PR[GP1:91,2] = PR[GP1:90,2] + 13.787;
   1:L PR[91] 10mm/sec CNT100;
   1:  PR[GP1:91,1] = PR[GP1:90,1] + 26.120;
   1:  PR[GP1:91,2] = PR[GP1:90,2] + 15.327;
   1:L PR[91] 10mm/sec CNT100;
   1:  PR[GP1:91,1] = PR[GP1:90,1] + 22.877;
   1:  PR[GP1:91,2] = PR[GP1:90,2] + 16.256;
   1:L PR[91] 10mm/sec CNT100;
   1:  PR[GP1:91,1] = PR[GP1:90,1] + 19.510;
   1:  PR[GP1:91,2] = PR[GP1:90,2] + 16.538;
   1:L PR[91] 10mm/sec CNT100;
   1:  PR[GP1:91,1] = PR[GP1:90,1] + 16.154;
   1:  PR[GP1:91,2] = PR[GP1:90,2] + 16.163;
   1:L PR[91] 10mm/sec CNT100;
   1:  PR[GP1:91,1] = PR[GP1:90,1] + 12.917;
   1:  PR[GP1:91,2] = PR[GP1:90,2] + 15.142;
   1:L PR[91] 10mm/sec CNT100;
   1:  PR[GP1:91,1] = PR[GP1:90,1] + 9.875;
   1:  PR[GP1:91,2] = PR[GP1:90,2] + 13.508;
   1:L PR[91] 10mm/sec CNT100;
   1:  PR[GP1:91,1] = PR[GP1:90,1] + 7.204;
   1:  PR[GP1:91,2] = PR[GP1:90,2] + 11.333;
   1:L PR[91] 10mm/sec CNT100;
   1:  PR[GP1:91,1] = PR[GP1:90,1] + 4.978;
   1:  PR[GP1:91,2] = PR[GP1:90,2] + 8.696;
   1:L PR[91] 10mm/sec CNT100;
   1:  PR[GP1:91,1] = PR[GP1:90,1] + 3.305;
   1:  PR[GP1:91,2] = PR[GP1:90,2] + 5.701;
   1:L PR[91] 10mm/sec CNT100;
   1:  PR[GP1:91,1] = PR[GP1:90,1] + 2.274;
   1:  PR[GP1:91,2] = PR[GP1:90,2] + 2.516;
   1:L PR[91] 10mm/sec CNT100;
   1:  PR[GP1:91,1] = PR[GP1:90,1] + 2.142;
   1:  PR[GP1:91,2] = PR[GP1:90,2] + 2.219;
   1:L PR[91] 10mm/sec CNT100;
   1:  PR[GP1:91,1] = PR[GP1:90,1] + 2.098;
   1:  PR[GP1:91,2] = PR[GP1:90,2] + 2.048;
   1:L PR[91] 10mm/sec CNT100;
   1:  PR[GP1:91,1] = PR[GP1:90,1] + 1.974;
   1:  PR[GP1:91,2] = PR[GP1:90,2] + 1.760;
   1:L PR[91] 10mm/sec CNT100;
   1:  PR[GP1:91,1] = PR[GP1:90,1] + 1.762;
   1:  PR[GP1:91,2] = PR[GP1:90,2] + 1.427;
   1:L PR[91] 10mm/sec CNT100;
   1:  PR[GP1:91,1] = PR[GP1:90,1] + 1.563;
   1:  PR[GP1:91,2] = PR[GP1:90,2] + 1.199;
   1:L PR[91] 10mm/sec CNT100;
   1:  PR[GP1:91,1] = PR[GP1:90,1] + 1.128;
   1:  PR[GP1:91,2] = PR[GP1:90,2] + 0.852;
   1:L PR[91] 10mm/sec CNT100;
   1:  PR[GP1:91,1] = PR[GP1:90,1] + 0.416;
   1:  PR[GP1:91,2] = PR[GP1:90,2] + 0.467;
   1:L PR[91] 10mm/sec CNT100;
   1:  PR[GP1:91,1] = PR[GP1:90,1] + -0.157;
   1:  PR[GP1:91,2] = PR[GP1:90,2] + 0.470;
   1:L PR[91] 10mm/sec CNT100;
   1:  PR[GP1:91,1] = PR[GP1:90,1] + -0.742;
   1:  PR[GP1:91,2] = PR[GP1:90,2] + 0.391;
   1:L PR[91] 10mm/sec CNT100;
   1:  PR[GP1:91,1] = PR[GP1:90,1] + -1.840;
   1:  PR[GP1:91,2] = PR[GP1:90,2] + 0.847;
   1:L PR[91] 10mm/sec CNT100;
   1:  PR[GP1:91,1] = PR[GP1:90,1] + -2.273;
   1:  PR[GP1:91,2] = PR[GP1:90,2] + 1.362;
   1:L PR[91] 10mm/sec CNT100;
   1:  PR[GP1:91,1] = PR[GP1:90,1] + -2.529;
   1:  PR[GP1:91,2] = PR[GP1:90,2] + 1.569;
   1:L PR[91] 10mm/sec CNT100;
   1:  PR[GP1:91,1] = PR[GP1:90,1] + -2.798;
   1:  PR[GP1:91,2] = PR[GP1:90,2] + 2.112;
   1:L PR[91] 10mm/sec CNT100;
   1:  PR[GP1:91,1] = PR[GP1:90,1] + -2.907;
   1:  PR[GP1:91,2] = PR[GP1:90,2] + 2.423;
   1:L PR[91] 10mm/sec CNT100;
   1:  PR[GP1:91,1] = PR[GP1:90,1] + -3.885;
   1:  PR[GP1:91,2] = PR[GP1:90,2] + 5.885;
   1:L PR[91] 10mm/sec CNT100;
   1:  PR[GP1:91,1] = PR[GP1:90,1] + -4.116;
   1:  PR[GP1:91,2] = PR[GP1:90,2] + 6.382;
   1:L PR[91] 10mm/sec CNT100;
   1:  PR[GP1:91,1] = PR[GP1:90,1] + -5.631;
   1:  PR[GP1:91,2] = PR[GP1:90,2] + 9.111;
   1:L PR[91] 10mm/sec CNT100;
   1:  PR[GP1:91,1] = PR[GP1:90,1] + -5.772;
   1:  PR[GP1:91,2] = PR[GP1:90,2] + 9.301;
   1:L PR[91] 10mm/sec CNT100;
   1:  PR[GP1:91,1] = PR[GP1:90,1] + -8.046;
   1:  PR[GP1:91,2] = PR[GP1:90,2] + 11.909;
   1:L PR[91] 10mm/sec CNT100;
   1:  PR[GP1:91,1] = PR[GP1:90,1] + -10.853;
   1:  PR[GP1:91,2] = PR[GP1:90,2] + 14.051;
   1:L PR[91] 10mm/sec CNT100;
   1:  PR[GP1:91,1] = PR[GP1:90,1] + -11.038;
   1:  PR[GP1:91,2] = PR[GP1:90,2] + 14.150;
   1:L PR[91] 10mm/sec CNT100;
   1:  PR[GP1:91,1] = PR[GP1:90,1] + -13.920;
   1:  PR[GP1:91,2] = PR[GP1:90,2] + 15.511;
   1:L PR[91] 10mm/sec CNT100;
   1:  PR[GP1:91,1] = PR[GP1:90,1] + -14.331;
   1:  PR[GP1:91,2] = PR[GP1:90,2] + 15.649;
   1:L PR[91] 10mm/sec CNT100;
   1:  PR[GP1:91,1] = PR[GP1:90,1] + -17.115;
   1:  PR[GP1:91,2] = PR[GP1:90,2] + 16.300;
   1:L PR[91] 10mm/sec CNT100;
   1:  PR[GP1:91,1] = PR[GP1:90,1] + -17.723;
   1:  PR[GP1:91,2] = PR[GP1:90,2] + 16.398;
   1:L PR[91] 10mm/sec CNT100;
   1:  PR[GP1:91,1] = PR[GP1:90,1] + -18.370;
   1:  PR[GP1:91,2] = PR[GP1:90,2] + 16.394;
   1:L PR[91] 10mm/sec CNT100;
   1:  PR[GP1:91,1] = PR[GP1:90,1] + -21.120;
   1:  PR[GP1:91,2] = PR[GP1:90,2] + 16.438;
   1:L PR[91] 10mm/sec CNT100;
   1:  PR[GP1:91,1] = PR[GP1:90,1] + -21.890;
   1:  PR[GP1:91,2] = PR[GP1:90,2] + 16.306;
   1:L PR[91] 10mm/sec CNT100;
   1:  PR[GP1:91,1] = PR[GP1:90,1] + -24.357;
   1:  PR[GP1:91,2] = PR[GP1:90,2] + 15.820;
   1:L PR[91] 10mm/sec CNT100;
   1:  PR[GP1:91,1] = PR[GP1:90,1] + -25.212;
   1:  PR[GP1:91,2] = PR[GP1:90,2] + 15.522;
   1:L PR[91] 10mm/sec CNT100;
   1:  PR[GP1:91,1] = PR[GP1:90,1] + -27.358;
   1:  PR[GP1:91,2] = PR[GP1:90,2] + 14.600;
   1:L PR[91] 10mm/sec CNT100;
   1:  PR[GP1:91,1] = PR[GP1:90,1] + -28.237;
   1:  PR[GP1:91,2] = PR[GP1:90,2] + 14.120;
   1:L PR[91] 10mm/sec CNT100;
   1:  PR[GP1:91,1] = PR[GP1:90,1] + -30.037;
   1:  PR[GP1:91,2] = PR[GP1:90,2] + 12.842;
   1:L PR[91] 10mm/sec CNT100;
   1:  PR[GP1:91,1] = PR[GP1:90,1] + -30.880;
   1:  PR[GP1:91,2] = PR[GP1:90,2] + 12.181;
   1:L PR[91] 10mm/sec CNT100;
   1:  PR[GP1:91,1] = PR[GP1:90,1] + -33.079;
   1:  PR[GP1:91,2] = PR[GP1:90,2] + 9.777;
   1:L PR[91] 10mm/sec CNT100;
   1:  PR[GP1:91,1] = PR[GP1:90,1] + -33.688;
   1:  PR[GP1:91,2] = PR[GP1:90,2] + 8.841;
   1:L PR[91] 10mm/sec CNT100;
   1:  PR[GP1:91,1] = PR[GP1:90,1] + -34.753;
   1:  PR[GP1:91,2] = PR[GP1:90,2] + 7.020;
   1:L PR[91] 10mm/sec CNT100;
   1:  PR[GP1:91,1] = PR[GP1:90,1] + -35.209;
   1:  PR[GP1:91,2] = PR[GP1:90,2] + 5.974;
   1:L PR[91] 10mm/sec CNT100;
   1:  PR[GP1:91,1] = PR[GP1:90,1] + -35.863;
   1:  PR[GP1:91,2] = PR[GP1:90,2] + 3.991;
   1:L PR[91] 10mm/sec CNT100;
   1:  PR[GP1:91,1] = PR[GP1:90,1] + -36.141;
   1:  PR[GP1:91,2] = PR[GP1:90,2] + 2.892;
   1:L PR[91] 10mm/sec CNT100;
   1:  PR[GP1:91,1] = PR[GP1:90,1] + -36.237;
   1:  PR[GP1:91,2] = PR[GP1:90,2] + 1.731;
   1:L PR[91] 10mm/sec CNT100;
   1:  PR[GP1:91,1] = PR[GP1:90,1] + -36.455;
   1:  PR[GP1:91,2] = PR[GP1:90,2] + -0.346;
   1:L PR[91] 10mm/sec CNT100;
   1:  PR[GP1:91,1] = PR[GP1:90,1] + -36.363;
   1:  PR[GP1:91,2] = PR[GP1:90,2] + -1.462;
   1:L PR[91] 10mm/sec CNT100;
   1:  PR[GP1:91,1] = PR[GP1:90,1] + -36.134;
   1:  PR[GP1:91,2] = PR[GP1:90,2] + -3.582;
   1:L PR[91] 10mm/sec CNT100;
   1:  PR[GP1:91,1] = PR[GP1:90,1] + -35.870;
   1:  PR[GP1:91,2] = PR[GP1:90,2] + -4.628;
   1:L PR[91] 10mm/sec CNT100;
   1:  PR[GP1:91,1] = PR[GP1:90,1] + -35.179;
   1:  PR[GP1:91,2] = PR[GP1:90,2] + -6.725;
   1:L PR[91] 10mm/sec CNT100;
   1:  PR[GP1:91,1] = PR[GP1:90,1] + -34.774;
   1:  PR[GP1:91,2] = PR[GP1:90,2] + -7.653;
   1:L PR[91] 10mm/sec CNT100;
   1:  PR[GP1:91,1] = PR[GP1:90,1] + -33.590;
   1:  PR[GP1:91,2] = PR[GP1:90,2] + -9.668;
   1:L PR[91] 10mm/sec CNT100;
   1:  PR[GP1:91,1] = PR[GP1:90,1] + -33.088;
   1:  PR[GP1:91,2] = PR[GP1:90,2] + -10.440;
   1:L PR[91] 10mm/sec CNT100;
   1:  PR[GP1:91,1] = PR[GP1:90,1] + -30.836;
   1:  PR[GP1:91,2] = PR[GP1:90,2] + -12.894;
   1:L PR[91] 10mm/sec CNT100;
   1:  PR[GP1:91,1] = PR[GP1:90,1] + -30.207;
   1:  PR[GP1:91,2] = PR[GP1:90,2] + -13.387;
   1:L PR[91] 10mm/sec CNT100;
   1:  PR[GP1:91,1] = PR[GP1:90,1] + -28.085;
   1:  PR[GP1:91,2] = PR[GP1:90,2] + -14.885;
   1:L PR[91] 10mm/sec CNT100;
   1:  PR[GP1:91,1] = PR[GP1:90,1] + -27.517;
   1:  PR[GP1:91,2] = PR[GP1:90,2] + -15.196;
   1:L PR[91] 10mm/sec CNT100;
   1:  PR[GP1:91,1] = PR[GP1:90,1] + -24.884;
   1:  PR[GP1:91,2] = PR[GP1:90,2] + -16.317;
   1:L PR[91] 10mm/sec CNT100;
   1:  PR[GP1:91,1] = PR[GP1:90,1] + -24.454;
   1:  PR[GP1:91,2] = PR[GP1:90,2] + -16.467;
   1:L PR[91] 10mm/sec CNT100;
   1:  PR[GP1:91,1] = PR[GP1:90,1] + -21.052;
   1:  PR[GP1:91,2] = PR[GP1:90,2] + -17.148;
   1:  PR[GP1:91,3] = PR[GP1:90,3] + 9.900;
   1:L PR[91] 10mm/sec CNT100;
   1:  PR[GP1:91,1] = PR[GP1:90,1] + -20.652;
   1:  PR[GP1:91,2] = PR[GP1:90,2] + -17.171;
   1:L PR[91] 10mm/sec CNT100;
   1:  PR[GP1:91,1] = PR[GP1:90,1] + -17.599;
   1:  PR[GP1:91,2] = PR[GP1:90,2] + -17.134;
   1:L PR[91] 10mm/sec CNT100;
   1:  PR[GP1:91,1] = PR[GP1:90,1] + -16.800;
   1:  PR[GP1:91,2] = PR[GP1:90,2] + -17.019;
   1:L PR[91] 10mm/sec CNT100;
   1:  PR[GP1:91,1] = PR[GP1:90,1] + -14.274;
   1:  PR[GP1:91,2] = PR[GP1:90,2] + -16.449;
   1:L PR[91] 10mm/sec CNT100;
   1:  PR[GP1:91,1] = PR[GP1:90,1] + -13.116;
   1:  PR[GP1:91,2] = PR[GP1:90,2] + -16.036;
   1:L PR[91] 10mm/sec CNT100;
   1:  PR[GP1:91,1] = PR[GP1:90,1] + -11.200;
   1:  PR[GP1:91,2] = PR[GP1:90,2] + -15.150;
   1:L PR[91] 10mm/sec CNT100;
   1:  PR[GP1:91,1] = PR[GP1:90,1] + -9.794;
   1:  PR[GP1:91,2] = PR[GP1:90,2] + -14.299;
   1:L PR[91] 10mm/sec CNT100;
   1:  PR[GP1:91,1] = PR[GP1:90,1] + -8.473;
   1:  PR[GP1:91,2] = PR[GP1:90,2] + -13.303;
   1:L PR[91] 10mm/sec CNT100;
   1:  PR[GP1:91,1] = PR[GP1:90,1] + -6.996;
   1:  PR[GP1:91,2] = PR[GP1:90,2] + -11.937;
   1:L PR[91] 10mm/sec CNT100;
   1:  PR[GP1:91,1] = PR[GP1:90,1] + -6.168;
   1:  PR[GP1:91,2] = PR[GP1:90,2] + -10.973;
   1:L PR[91] 10mm/sec CNT100;
   1:  PR[GP1:91,1] = PR[GP1:90,1] + -4.832;
   1:  PR[GP1:91,2] = PR[GP1:90,2] + -9.102;
   1:L PR[91] 10mm/sec CNT100;
   1:  PR[GP1:91,1] = PR[GP1:90,1] + -4.352;
   1:  PR[GP1:91,2] = PR[GP1:90,2] + -8.212;
   1:L PR[91] 10mm/sec CNT100;
   1:  PR[GP1:91,1] = PR[GP1:90,1] + -3.350;
   1:  PR[GP1:91,2] = PR[GP1:90,2] + -5.961;
   1:L PR[91] 10mm/sec CNT100;
   1:  PR[GP1:91,1] = PR[GP1:90,1] + -3.116;
   1:  PR[GP1:91,2] = PR[GP1:90,2] + -5.146;
   1:L PR[91] 10mm/sec CNT100;
   1:  PR[GP1:91,1] = PR[GP1:90,1] + -3.065;
   1:  PR[GP1:91,2] = PR[GP1:90,2] + -4.884;
   1:L PR[91] 10mm/sec CNT100;
   1:  PR[GP1:91,1] = PR[GP1:90,1] + -2.781;
   1:  PR[GP1:91,2] = PR[GP1:90,2] + -4.145;
   1:L PR[91] 10mm/sec CNT100;
   1:  PR[GP1:91,1] = PR[GP1:90,1] + -2.652;
   1:  PR[GP1:91,2] = PR[GP1:90,2] + -3.757;
   1:L PR[91] 10mm/sec CNT100;
   1:  PR[GP1:91,1] = PR[GP1:90,1] + -2.418;
   1:  PR[GP1:91,2] = PR[GP1:90,2] + -3.325;
   1:L PR[91] 10mm/sec CNT100;
   1:  PR[GP1:91,1] = PR[GP1:90,1] + -2.201;
   1:  PR[GP1:91,2] = PR[GP1:90,2] + -3.155;
   1:L PR[91] 10mm/sec CNT100;
   1:  PR[GP1:91,1] = PR[GP1:90,1] + -1.416;
   1:  PR[GP1:91,2] = PR[GP1:90,2] + -2.324;
   1:L PR[91] 10mm/sec CNT100;
   1:  PR[GP1:91,1] = PR[GP1:90,1] + 0.035;
   1:  PR[GP1:91,2] = PR[GP1:90,2] + -2.063;
   1:L PR[91] 10mm/sec CNT100;
   1:  PR[GP1:91,1] = PR[GP1:90,1] + 1.245;
   1:  PR[GP1:91,2] = PR[GP1:90,2] + -2.898;
   1:L PR[91] 10mm/sec CNT100;
   1:  PR[GP1:91,1] = PR[GP1:90,1] + 1.407;
   1:  PR[GP1:91,2] = PR[GP1:90,2] + -3.191;
   1:L PR[91] 10mm/sec CNT100;
   1:  PR[GP1:91,1] = PR[GP1:90,1] + 1.585;
   1:  PR[GP1:91,2] = PR[GP1:90,2] + -3.720;
   1:L PR[91] 10mm/sec CNT100;
   1:  PR[GP1:91,1] = PR[GP1:90,1] + 1.875;
   1:  PR[GP1:91,2] = PR[GP1:90,2] + -4.439;
   1:L PR[91] 10mm/sec CNT100;
   1:  PR[GP1:91,1] = PR[GP1:90,1] + 2.064;
   1:  PR[GP1:91,2] = PR[GP1:90,2] + -5.179;
   1:L PR[91] 10mm/sec CNT100;
   1:  PR[GP1:91,1] = PR[GP1:90,1] + 2.331;
   1:  PR[GP1:91,2] = PR[GP1:90,2] + -6.039;
   1:L PR[91] 10mm/sec CNT100;
   1:  PR[GP1:91,1] = PR[GP1:90,1] + 3.210;
   1:  PR[GP1:91,2] = PR[GP1:90,2] + -7.987;
   1:L PR[91] 10mm/sec CNT100;
   1:  PR[GP1:91,1] = PR[GP1:90,1] + 3.470;
   1:  PR[GP1:91,2] = PR[GP1:90,2] + -8.499;
   1:L PR[91] 10mm/sec CNT100;
   1:  PR[GP1:91,1] = PR[GP1:90,1] + 4.820;
   1:  PR[GP1:91,2] = PR[GP1:90,2] + -10.474;
   1:L PR[91] 10mm/sec CNT100;
   1:  PR[GP1:91,1] = PR[GP1:90,1] + 4.946;
   1:  PR[GP1:91,2] = PR[GP1:90,2] + -10.644;
   1:L PR[91] 10mm/sec CNT100;
   1:  PR[GP1:91,1] = PR[GP1:90,1] + 6.811;
   1:  PR[GP1:91,2] = PR[GP1:90,2] + -12.597;
   1:L PR[91] 10mm/sec CNT100;
   1:  PR[GP1:91,1] = PR[GP1:90,1] + 9.024;
   1:  PR[GP1:91,2] = PR[GP1:90,2] + -14.285;
   1:L PR[91] 10mm/sec CNT100;
   1:  PR[GP1:91,1] = PR[GP1:90,1] + 11.499;
   1:  PR[GP1:91,2] = PR[GP1:90,2] + -15.615;
   1:L PR[91] 10mm/sec CNT100;
   1:  PR[GP1:91,1] = PR[GP1:90,1] + 12.517;
   1:  PR[GP1:91,2] = PR[GP1:90,2] + -15.974;
   1:L PR[91] 10mm/sec CNT100;
   1:  PR[GP1:91,1] = PR[GP1:90,1] + 14.130;
   1:  PR[GP1:91,2] = PR[GP1:90,2] + -16.570;
   1:L PR[91] 10mm/sec CNT100;
   1:  PR[GP1:91,1] = PR[GP1:90,1] + 16.842;
   1:  PR[GP1:91,2] = PR[GP1:90,2] + -17.125;
   1:L PR[91] 10mm/sec CNT100;
   1:  PR[GP1:91,1] = PR[GP1:90,1] + 19.608;
   1:  PR[GP1:91,2] = PR[GP1:90,2] + -17.267;
   1:L PR[91] 10mm/sec CNT100;
   1:  PR[GP1:91,1] = PR[GP1:90,1] + 22.306;
   1:  PR[GP1:91,2] = PR[GP1:90,2] + -17.010;
   1:L PR[91] 10mm/sec CNT100;
   1:  PR[GP1:91,1] = PR[GP1:90,1] + 24.905;
   1:  PR[GP1:91,2] = PR[GP1:90,2] + -16.355;
   1:L PR[91] 10mm/sec CNT100;
   1:  PR[GP1:91,1] = PR[GP1:90,1] + 27.369;
   1:  PR[GP1:91,2] = PR[GP1:90,2] + -15.313;
   1:L PR[91] 10mm/sec CNT100;
   1:  PR[GP1:91,1] = PR[GP1:90,1] + 29.640;
   1:  PR[GP1:91,2] = PR[GP1:90,2] + -13.910;
   1:L PR[91] 10mm/sec CNT100;
   1:  PR[GP1:91,1] = PR[GP1:90,1] + 31.662;
   1:  PR[GP1:91,2] = PR[GP1:90,2] + -12.179;
   1:L PR[91] 10mm/sec CNT100;
   1:  PR[GP1:91,1] = PR[GP1:90,1] + 33.388;
   1:  PR[GP1:91,2] = PR[GP1:90,2] + -10.162;
   1:L PR[91] 10mm/sec CNT100;
   1:  PR[GP1:91,1] = PR[GP1:90,1] + 34.776;
   1:  PR[GP1:91,2] = PR[GP1:90,2] + -7.908;
   1:L PR[91] 10mm/sec CNT100;
   1:  PR[GP1:91,1] = PR[GP1:90,1] + 35.793;
   1:  PR[GP1:91,2] = PR[GP1:90,2] + -5.472;
   1:L PR[91] 10mm/sec CNT100;
   1:  PR[GP1:91,1] = PR[GP1:90,1] + 36.414;
   1:  PR[GP1:91,2] = PR[GP1:90,2] + -2.912;
   1:L PR[91] 10mm/sec CNT100;
   1:  PR[GP1:91,1] = PR[GP1:90,1] + 36.627;
   1:  PR[GP1:91,2] = PR[GP1:90,2] + -0.300;
   1:L PR[91] 10mm/sec CNT100;
   1:  PR[GP1:91,1] = PR[GP1:90,1] + 36.276;
   1:  PR[GP1:91,2] = PR[GP1:90,2] + 3.013;
   1:L PR[91] 10mm/sec CNT100;
   1:  PR[GP1:91,1] = PR[GP1:90,1] + 35.292;
   1:  PR[GP1:91,2] = PR[GP1:90,2] + 6.196;
   1:L PR[91] 10mm/sec CNT100;
   1:  PR[GP1:91,1] = PR[GP1:90,1] + 33.693;
   1:  PR[GP1:91,2] = PR[GP1:90,2] + 9.123;
   1:L PR[91] 10mm/sec CNT100;
   1:  PR[GP1:91,1] = PR[GP1:90,1] + 31.538;
   1:  PR[GP1:91,2] = PR[GP1:90,2] + 11.681;
   1:L PR[91] 10mm/sec CNT100;
   1:  PR[GP1:91,1] = PR[GP1:90,1] + 28.914;
   1:  PR[GP1:91,2] = PR[GP1:90,2] + 13.771;
   1:L PR[91] 10mm/sec CNT100;
   1:  PR[GP1:91,1] = PR[GP1:90,1] + 25.922;
   1:  PR[GP1:91,2] = PR[GP1:90,2] + 15.310;
   1:L PR[91] 10mm/sec CNT100;
   1:  PR[GP1:91,1] = PR[GP1:90,1] + 22.682;
   1:  PR[GP1:91,2] = PR[GP1:90,2] + 16.239;
   1:L PR[91] 10mm/sec CNT100;
   1:  PR[GP1:91,1] = PR[GP1:90,1] + 19.306;
   1:  PR[GP1:91,2] = PR[GP1:90,2] + 16.520;
   1:L PR[91] 10mm/sec CNT100;
   1:  PR[GP1:91,1] = PR[GP1:90,1] + 15.905;
   1:  PR[GP1:91,2] = PR[GP1:90,2] + 16.139;
   1:L PR[91] 10mm/sec CNT100;
   1:  PR[GP1:91,1] = PR[GP1:90,1] + 12.593;
   1:  PR[GP1:91,2] = PR[GP1:90,2] + 15.108;
   1:L PR[91] 10mm/sec CNT100;
   1:  PR[GP1:91,1] = PR[GP1:90,1] + 9.526;
   1:  PR[GP1:91,2] = PR[GP1:90,2] + 13.471;
   1:L PR[91] 10mm/sec CNT100;
   1:  PR[GP1:91,1] = PR[GP1:90,1] + 6.795;
   1:  PR[GP1:91,2] = PR[GP1:90,2] + 11.286;
   1:L PR[91] 10mm/sec CNT100;
   1:  PR[GP1:91,1] = PR[GP1:90,1] + 4.519;
   1:  PR[GP1:91,2] = PR[GP1:90,2] + 8.639;
   1:L PR[91] 10mm/sec CNT100;
   1:  PR[GP1:91,1] = PR[GP1:90,1] + 2.826;
   1:  PR[GP1:91,2] = PR[GP1:90,2] + 5.641;
   1:L PR[91] 10mm/sec CNT100;
   1:  PR[GP1:91,1] = PR[GP1:90,1] + 1.954;
   1:  PR[GP1:91,2] = PR[GP1:90,2] + 3.005;
   1:L PR[91] 10mm/sec CNT100;
   1:  PR[GP1:91,1] = PR[GP1:90,1] + 1.290;
   1:  PR[GP1:91,2] = PR[GP1:90,2] + 1.784;
   1:L PR[91] 10mm/sec CNT100;
   1:  PR[GP1:91,1] = PR[GP1:90,1] + 0.463;
   1:  PR[GP1:91,2] = PR[GP1:90,2] + 1.268;
   1:L PR[91] 10mm/sec CNT100;
   1:  PR[GP1:91,1] = PR[GP1:90,1] + -0.112;
   1:  PR[GP1:91,2] = PR[GP1:90,2] + 1.057;
   1:L PR[91] 10mm/sec CNT100;
   1:  PR[GP1:91,1] = PR[GP1:90,1] + -0.982;
   1:  PR[GP1:91,2] = PR[GP1:90,2] + 1.185;
   1:L PR[91] 10mm/sec CNT100;
   1:  PR[GP1:91,1] = PR[GP1:90,1] + -1.441;
   1:  PR[GP1:91,2] = PR[GP1:90,2] + 1.325;
   1:L PR[91] 10mm/sec CNT100;
   1:  PR[GP1:91,1] = PR[GP1:90,1] + -2.487;
   1:  PR[GP1:91,2] = PR[GP1:90,2] + 2.334;
   1:L PR[91] 10mm/sec CNT100;
   1:  PR[GP1:91,1] = PR[GP1:90,1] + -3.006;
   1:  PR[GP1:91,2] = PR[GP1:90,2] + 3.554;
   1:L PR[91] 10mm/sec CNT100;
   1:  PR[GP1:91,1] = PR[GP1:90,1] + -3.562;
   1:  PR[GP1:91,2] = PR[GP1:90,2] + 5.514;
   1:L PR[91] 10mm/sec CNT100;
   1:  PR[GP1:91,1] = PR[GP1:90,1] + -4.227;
   1:  PR[GP1:91,2] = PR[GP1:90,2] + 6.944;
   1:L PR[91] 10mm/sec CNT100;
   1:  PR[GP1:91,1] = PR[GP1:90,1] + -5.222;
   1:  PR[GP1:91,2] = PR[GP1:90,2] + 8.737;
   1:L PR[91] 10mm/sec CNT100;
   1:  PR[GP1:91,1] = PR[GP1:90,1] + -5.939;
   1:  PR[GP1:91,2] = PR[GP1:90,2] + 9.705;
   1:L PR[91] 10mm/sec CNT100;
   1:  PR[GP1:91,1] = PR[GP1:90,1] + -7.591;
   1:  PR[GP1:91,2] = PR[GP1:90,2] + 11.595;
   1:L PR[91] 10mm/sec CNT100;
   1:  PR[GP1:91,1] = PR[GP1:90,1] + -8.187;
   1:  PR[GP1:91,2] = PR[GP1:90,2] + 12.134;
   1:L PR[91] 10mm/sec CNT100;
   1:  PR[GP1:91,1] = PR[GP1:90,1] + -10.552;
   1:  PR[GP1:91,2] = PR[GP1:90,2] + 13.906;
   1:L PR[91] 10mm/sec CNT100;
   1:  PR[GP1:91,1] = PR[GP1:90,1] + -10.915;
   1:  PR[GP1:91,2] = PR[GP1:90,2] + 14.122;
   1:L PR[91] 10mm/sec CNT100;
   1:  PR[GP1:91,1] = PR[GP1:90,1] + -13.968;
   1:  PR[GP1:91,2] = PR[GP1:90,2] + 15.538;
   1:L PR[91] 10mm/sec CNT100;
   1:  PR[GP1:91,1] = PR[GP1:90,1] + -14.036;
   1:  PR[GP1:91,2] = PR[GP1:90,2] + 15.562;
   1:L PR[91] 10mm/sec CNT100;
   1:  PR[GP1:91,1] = PR[GP1:90,1] + -17.533;
   1:  PR[GP1:91,2] = PR[GP1:90,2] + 16.365;
   1:L PR[91] 10mm/sec CNT100;
   1:  PR[GP1:91,1] = PR[GP1:90,1] + -21.053;
   1:  PR[GP1:91,2] = PR[GP1:90,2] + 16.419;
   1:L PR[91] 10mm/sec CNT100;
   1:  PR[GP1:91,1] = PR[GP1:90,1] + -24.433;
   1:  PR[GP1:91,2] = PR[GP1:90,2] + 15.761;
   1:L PR[91] 10mm/sec CNT100;
   1:  PR[GP1:91,1] = PR[GP1:90,1] + -24.822;
   1:  PR[GP1:91,2] = PR[GP1:90,2] + 15.626;
   1:L PR[91] 10mm/sec CNT100;
   1:  PR[GP1:91,1] = PR[GP1:90,1] + -27.537;
   1:  PR[GP1:91,2] = PR[GP1:90,2] + 14.460;
   1:L PR[91] 10mm/sec CNT100;
   1:  PR[GP1:91,1] = PR[GP1:90,1] + -28.004;
   1:  PR[GP1:91,2] = PR[GP1:90,2] + 14.204;
   1:L PR[91] 10mm/sec CNT100;
   1:  PR[GP1:91,1] = PR[GP1:90,1] + -30.282;
   1:  PR[GP1:91,2] = PR[GP1:90,2] + 12.586;
   1:L PR[91] 10mm/sec CNT100;
   1:  PR[GP1:91,1] = PR[GP1:90,1] + -30.770;
   1:  PR[GP1:91,2] = PR[GP1:90,2] + 12.203;
   1:L PR[91] 10mm/sec CNT100;
   1:  PR[GP1:91,1] = PR[GP1:90,1] + -33.054;
   1:  PR[GP1:91,2] = PR[GP1:90,2] + 9.706;
   1:L PR[91] 10mm/sec CNT100;
   1:  PR[GP1:91,1] = PR[GP1:90,1] + -33.424;
   1:  PR[GP1:91,2] = PR[GP1:90,2] + 9.137;
   1:L PR[91] 10mm/sec CNT100;
   1:  PR[GP1:91,1] = PR[GP1:90,1] + -34.771;
   1:  PR[GP1:91,2] = PR[GP1:90,2] + 6.832;
   1:L PR[91] 10mm/sec CNT100;
   1:  PR[GP1:91,1] = PR[GP1:90,1] + -35.055;
   1:  PR[GP1:91,2] = PR[GP1:90,2] + 6.183;
   1:L PR[91] 10mm/sec CNT100;
   1:  PR[GP1:91,1] = PR[GP1:90,1] + -35.883;
   1:  PR[GP1:91,2] = PR[GP1:90,2] + 3.673;
   1:L PR[91] 10mm/sec CNT100;
   1:  PR[GP1:91,1] = PR[GP1:90,1] + -36.055;
   1:  PR[GP1:91,2] = PR[GP1:90,2] + 2.992;
   1:L PR[91] 10mm/sec CNT100;
   1:  PR[GP1:91,1] = PR[GP1:90,1] + -36.115;
   1:  PR[GP1:91,2] = PR[GP1:90,2] + 2.261;
   1:L PR[91] 10mm/sec CNT100;
   1:  PR[GP1:91,1] = PR[GP1:90,1] + -36.391;
   1:  PR[GP1:91,2] = PR[GP1:90,2] + -0.367;
   1:L PR[91] 10mm/sec CNT100;
   1:  PR[GP1:91,1] = PR[GP1:90,1] + -36.335;
   1:  PR[GP1:91,2] = PR[GP1:90,2] + -1.046;
   1:L PR[91] 10mm/sec CNT100;
   1:  PR[GP1:91,1] = PR[GP1:90,1] + -36.045;
   1:  PR[GP1:91,2] = PR[GP1:90,2] + -3.729;
   1:L PR[91] 10mm/sec CNT100;
   1:  PR[GP1:91,1] = PR[GP1:90,1] + -35.891;
   1:  PR[GP1:91,2] = PR[GP1:90,2] + -4.341;
   1:L PR[91] 10mm/sec CNT100;
   1:  PR[GP1:91,1] = PR[GP1:90,1] + -35.017;
   1:  PR[GP1:91,2] = PR[GP1:90,2] + -6.994;
   1:L PR[91] 10mm/sec CNT100;
   1:  PR[GP1:91,1] = PR[GP1:90,1] + -34.798;
   1:  PR[GP1:91,2] = PR[GP1:90,2] + -7.496;
   1:L PR[91] 10mm/sec CNT100;
   1:  PR[GP1:91,1] = PR[GP1:90,1] + -33.300;
   1:  PR[GP1:91,2] = PR[GP1:90,2] + -10.044;
   1:L PR[91] 10mm/sec CNT100;
   1:  PR[GP1:91,1] = PR[GP1:90,1] + -33.065;
   1:  PR[GP1:91,2] = PR[GP1:90,2] + -10.406;
   1:L PR[91] 10mm/sec CNT100;
   1:  PR[GP1:91,1] = PR[GP1:90,1] + -30.715;
   1:  PR[GP1:91,2] = PR[GP1:90,2] + -12.966;
   1:L PR[91] 10mm/sec CNT100;
   1:  PR[GP1:91,1] = PR[GP1:90,1] + -30.495;
   1:  PR[GP1:91,2] = PR[GP1:90,2] + -13.138;
   1:L PR[91] 10mm/sec CNT100;
   1:  PR[GP1:91,1] = PR[GP1:90,1] + -27.813;
   1:  PR[GP1:91,2] = PR[GP1:90,2] + -15.033;
   1:L PR[91] 10mm/sec CNT100;
   1:  PR[GP1:91,1] = PR[GP1:90,1] + -27.736;
   1:  PR[GP1:91,2] = PR[GP1:90,2] + -15.076;
   1:L PR[91] 10mm/sec CNT100;
   1:  PR[GP1:91,1] = PR[GP1:90,1] + -24.511;
   1:  PR[GP1:91,2] = PR[GP1:90,2] + -16.452;
   1:L PR[91] 10mm/sec CNT100;
   1:  PR[GP1:91,1] = PR[GP1:90,1] + -23.679;
   1:  PR[GP1:91,2] = PR[GP1:90,2] + -16.671;
   1:  PR[GP1:91,3] = PR[GP1:90,3] + 11.000;
   1:L PR[91] 10mm/sec CNT100;
   1:  PR[GP1:91,1] = PR[GP1:90,1] + -21.131;
   1:  PR[GP1:91,2] = PR[GP1:90,2] + -17.179;
   1:L PR[91] 10mm/sec CNT100;
   1:  PR[GP1:91,1] = PR[GP1:90,1] + -19.847;
   1:  PR[GP1:91,2] = PR[GP1:90,2] + -17.252;
   1:L PR[91] 10mm/sec CNT100;
   1:  PR[GP1:91,1] = PR[GP1:90,1] + -17.744;
   1:  PR[GP1:91,2] = PR[GP1:90,2] + -17.227;
   1:L PR[91] 10mm/sec CNT100;
   1:  PR[GP1:91,1] = PR[GP1:90,1] + -16.002;
   1:  PR[GP1:91,2] = PR[GP1:90,2] + -16.977;
   1:L PR[91] 10mm/sec CNT100;
   1:  PR[GP1:91,1] = PR[GP1:90,1] + -14.479;
   1:  PR[GP1:91,2] = PR[GP1:90,2] + -16.633;
   1:L PR[91] 10mm/sec CNT100;
   1:  PR[GP1:91,1] = PR[GP1:90,1] + -12.358;
   1:  PR[GP1:91,2] = PR[GP1:90,2] + -15.876;
   1:L PR[91] 10mm/sec CNT100;
   1:  PR[GP1:91,1] = PR[GP1:90,1] + -11.447;
   1:  PR[GP1:91,2] = PR[GP1:90,2] + -15.455;
   1:L PR[91] 10mm/sec CNT100;
   1:  PR[GP1:91,1] = PR[GP1:90,1] + -9.108;
   1:  PR[GP1:91,2] = PR[GP1:90,2] + -14.040;
   1:L PR[91] 10mm/sec CNT100;
   1:  PR[GP1:91,1] = PR[GP1:90,1] + -8.732;
   1:  PR[GP1:91,2] = PR[GP1:90,2] + -13.757;
   1:L PR[91] 10mm/sec CNT100;
   1:  PR[GP1:91,1] = PR[GP1:90,1] + -6.429;
   1:  PR[GP1:91,2] = PR[GP1:90,2] + -11.626;
   1:L PR[91] 10mm/sec CNT100;
   1:  PR[GP1:91,1] = PR[GP1:90,1] + -4.456;
   1:  PR[GP1:91,2] = PR[GP1:90,2] + -8.927;
   1:L PR[91] 10mm/sec CNT100;
   1:  PR[GP1:91,1] = PR[GP1:90,1] + -4.378;
   1:  PR[GP1:91,2] = PR[GP1:90,2] + -8.808;
   1:L PR[91] 10mm/sec CNT100;
   1:  PR[GP1:91,1] = PR[GP1:90,1] + -3.125;
   1:  PR[GP1:91,2] = PR[GP1:90,2] + -6.065;
   1:L PR[91] 10mm/sec CNT100;
   1:  PR[GP1:91,1] = PR[GP1:90,1] + -2.949;
   1:  PR[GP1:91,2] = PR[GP1:90,2] + -5.534;
   1:L PR[91] 10mm/sec CNT100;
   1:  PR[GP1:91,1] = PR[GP1:90,1] + -2.473;
   1:  PR[GP1:91,2] = PR[GP1:90,2] + -4.659;
   1:L PR[91] 10mm/sec CNT100;
   1:  PR[GP1:91,1] = PR[GP1:90,1] + -2.006;
   1:  PR[GP1:91,2] = PR[GP1:90,2] + -4.291;
   1:L PR[91] 10mm/sec CNT100;
   1:  PR[GP1:91,1] = PR[GP1:90,1] + -1.478;
   1:  PR[GP1:91,2] = PR[GP1:90,2] + -3.732;
   1:L PR[91] 10mm/sec CNT100;
   1:  PR[GP1:91,1] = PR[GP1:90,1] + -0.899;
   1:  PR[GP1:91,2] = PR[GP1:90,2] + -3.676;
   1:L PR[91] 10mm/sec CNT100;
   1:  PR[GP1:91,1] = PR[GP1:90,1] + -0.108;
   1:  PR[GP1:91,2] = PR[GP1:90,2] + -3.537;
   1:L PR[91] 10mm/sec CNT100;
   1:  PR[GP1:91,1] = PR[GP1:90,1] + 1.055;
   1:  PR[GP1:91,2] = PR[GP1:90,2] + -4.312;
   1:L PR[91] 10mm/sec CNT100;
   1:  PR[GP1:91,1] = PR[GP1:90,1] + 1.460;
   1:  PR[GP1:91,2] = PR[GP1:90,2] + -5.045;
   1:L PR[91] 10mm/sec CNT100;
   1:  PR[GP1:91,1] = PR[GP1:90,1] + 1.852;
   1:  PR[GP1:91,2] = PR[GP1:90,2] + -6.284;
   1:L PR[91] 10mm/sec CNT100;
   1:  PR[GP1:91,1] = PR[GP1:90,1] + 2.349;
   1:  PR[GP1:91,2] = PR[GP1:90,2] + -7.411;
   1:L PR[91] 10mm/sec CNT100;
   1:  PR[GP1:91,1] = PR[GP1:90,1] + 3.074;
   1:  PR[GP1:91,2] = PR[GP1:90,2] + -8.838;
   1:L PR[91] 10mm/sec CNT100;
   1:  PR[GP1:91,1] = PR[GP1:90,1] + 3.803;
   1:  PR[GP1:91,2] = PR[GP1:90,2] + -9.904;
   1:L PR[91] 10mm/sec CNT100;
   1:  PR[GP1:91,1] = PR[GP1:90,1] + 4.579;
   1:  PR[GP1:91,2] = PR[GP1:90,2] + -10.951;
   1:L PR[91] 10mm/sec CNT100;
   1:  PR[GP1:91,1] = PR[GP1:90,1] + 5.846;
   1:  PR[GP1:91,2] = PR[GP1:90,2] + -12.261;
   1:L PR[91] 10mm/sec CNT100;
   1:  PR[GP1:91,1] = PR[GP1:90,1] + 6.412;
   1:  PR[GP1:91,2] = PR[GP1:90,2] + -12.808;
   1:L PR[91] 10mm/sec CNT100;
   1:  PR[GP1:91,1] = PR[GP1:90,1] + 8.544;
   1:  PR[GP1:91,2] = PR[GP1:90,2] + -14.387;
   1:L PR[91] 10mm/sec CNT100;
   1:  PR[GP1:91,1] = PR[GP1:90,1] + 11.022;
   1:  PR[GP1:91,2] = PR[GP1:90,2] + -15.716;
   1:L PR[91] 10mm/sec CNT100;
   1:  PR[GP1:91,1] = PR[GP1:90,1] + 13.707;
   1:  PR[GP1:91,2] = PR[GP1:90,2] + -16.664;
   1:L PR[91] 10mm/sec CNT100;
   1:  PR[GP1:91,1] = PR[GP1:90,1] + 16.495;
   1:  PR[GP1:91,2] = PR[GP1:90,2] + -17.208;
   1:L PR[91] 10mm/sec CNT100;
   1:  PR[GP1:91,1] = PR[GP1:90,1] + 19.274;
   1:  PR[GP1:91,2] = PR[GP1:90,2] + -17.348;
   1:L PR[91] 10mm/sec CNT100;
   1:  PR[GP1:91,1] = PR[GP1:90,1] + 22.035;
   1:  PR[GP1:91,2] = PR[GP1:90,2] + -17.075;
   1:L PR[91] 10mm/sec CNT100;
   1:  PR[GP1:91,1] = PR[GP1:90,1] + 24.711;
   1:  PR[GP1:91,2] = PR[GP1:90,2] + -16.398;
   1:L PR[91] 10mm/sec CNT100;
   1:  PR[GP1:91,1] = PR[GP1:90,1] + 27.176;
   1:  PR[GP1:91,2] = PR[GP1:90,2] + -15.353;
   1:L PR[91] 10mm/sec CNT100;
   1:  PR[GP1:91,1] = PR[GP1:90,1] + 29.448;
   1:  PR[GP1:91,2] = PR[GP1:90,2] + -13.946;
   1:L PR[91] 10mm/sec CNT100;
   1:  PR[GP1:91,1] = PR[GP1:90,1] + 31.470;
   1:  PR[GP1:91,2] = PR[GP1:90,2] + -12.211;
   1:L PR[91] 10mm/sec CNT100;
   1:  PR[GP1:91,1] = PR[GP1:90,1] + 33.196;
   1:  PR[GP1:91,2] = PR[GP1:90,2] + -10.191;
   1:L PR[91] 10mm/sec CNT100;
   1:  PR[GP1:91,1] = PR[GP1:90,1] + 34.582;
   1:  PR[GP1:91,2] = PR[GP1:90,2] + -7.934;
   1:L PR[91] 10mm/sec CNT100;
   1:  PR[GP1:91,1] = PR[GP1:90,1] + 35.598;
   1:  PR[GP1:91,2] = PR[GP1:90,2] + -5.496;
   1:L PR[91] 10mm/sec CNT100;
   1:  PR[GP1:91,1] = PR[GP1:90,1] + 36.217;
   1:  PR[GP1:91,2] = PR[GP1:90,2] + -2.934;
   1:L PR[91] 10mm/sec CNT100;
   1:  PR[GP1:91,1] = PR[GP1:90,1] + 36.372;
   1:  PR[GP1:91,2] = PR[GP1:90,2] + -1.001;
   1:L PR[91] 10mm/sec CNT100;
   1:  PR[GP1:91,1] = PR[GP1:90,1] + 36.449;
   1:  PR[GP1:91,2] = PR[GP1:90,2] + -0.308;
   1:L PR[91] 10mm/sec CNT100;
   1:  PR[GP1:91,1] = PR[GP1:90,1] + 36.088;
   1:  PR[GP1:91,2] = PR[GP1:90,2] + 2.996;
   1:L PR[91] 10mm/sec CNT100;
   1:  PR[GP1:91,1] = PR[GP1:90,1] + 35.101;
   1:  PR[GP1:91,2] = PR[GP1:90,2] + 6.180;
   1:L PR[91] 10mm/sec CNT100;
   1:  PR[GP1:91,1] = PR[GP1:90,1] + 33.498;
   1:  PR[GP1:91,2] = PR[GP1:90,2] + 9.107;
   1:L PR[91] 10mm/sec CNT100;
   1:  PR[GP1:91,1] = PR[GP1:90,1] + 31.342;
   1:  PR[GP1:91,2] = PR[GP1:90,2] + 11.666;
   1:L PR[91] 10mm/sec CNT100;
   1:  PR[GP1:91,1] = PR[GP1:90,1] + 28.716;
   1:  PR[GP1:91,2] = PR[GP1:90,2] + 13.755;
   1:L PR[91] 10mm/sec CNT100;
   1:  PR[GP1:91,1] = PR[GP1:90,1] + 25.724;
   1:  PR[GP1:91,2] = PR[GP1:90,2] + 15.294;
   1:L PR[91] 10mm/sec CNT100;
   1:  PR[GP1:91,1] = PR[GP1:90,1] + 22.487;
   1:  PR[GP1:91,2] = PR[GP1:90,2] + 16.222;
   1:L PR[91] 10mm/sec CNT100;
   1:  PR[GP1:91,1] = PR[GP1:90,1] + 19.042;
   1:  PR[GP1:91,2] = PR[GP1:90,2] + 16.495;
   1:L PR[91] 10mm/sec CNT100;
   1:  PR[GP1:91,1] = PR[GP1:90,1] + 15.586;
   1:  PR[GP1:91,2] = PR[GP1:90,2] + 16.108;
   1:L PR[91] 10mm/sec CNT100;
   1:  PR[GP1:91,1] = PR[GP1:90,1] + 12.251;
   1:  PR[GP1:91,2] = PR[GP1:90,2] + 15.073;
   1:L PR[91] 10mm/sec CNT100;
   1:  PR[GP1:91,1] = PR[GP1:90,1] + 9.114;
   1:  PR[GP1:91,2] = PR[GP1:90,2] + 13.425;
   1:L PR[91] 10mm/sec CNT100;
   1:  PR[GP1:91,1] = PR[GP1:90,1] + 6.333;
   1:  PR[GP1:91,2] = PR[GP1:90,2] + 11.229;
   1:L PR[91] 10mm/sec CNT100;
   1:  PR[GP1:91,1] = PR[GP1:90,1] + 4.041;
   1:  PR[GP1:91,2] = PR[GP1:90,2] + 8.579;
   1:L PR[91] 10mm/sec CNT100;
   1:  PR[GP1:91,1] = PR[GP1:90,1] + 2.314;
   1:  PR[GP1:91,2] = PR[GP1:90,2] + 5.569;
   1:L PR[91] 10mm/sec CNT100;
   1:  PR[GP1:91,1] = PR[GP1:90,1] + 1.805;
   1:  PR[GP1:91,2] = PR[GP1:90,2] + 4.034;
   1:L PR[91] 10mm/sec CNT100;
   1:  PR[GP1:91,1] = PR[GP1:90,1] + 1.437;
   1:  PR[GP1:91,2] = PR[GP1:90,2] + 3.361;
   1:L PR[91] 10mm/sec CNT100;
   1:  PR[GP1:91,1] = PR[GP1:90,1] + 1.076;
   1:  PR[GP1:91,2] = PR[GP1:90,2] + 2.827;
   1:L PR[91] 10mm/sec CNT100;
   1:  PR[GP1:91,1] = PR[GP1:90,1] + 0.290;
   1:  PR[GP1:91,2] = PR[GP1:90,2] + 2.368;
   1:L PR[91] 10mm/sec CNT100;
   1:  PR[GP1:91,1] = PR[GP1:90,1] + -0.261;
   1:  PR[GP1:91,2] = PR[GP1:90,2] + 2.151;
   1:L PR[91] 10mm/sec CNT100;
   1:  PR[GP1:91,1] = PR[GP1:90,1] + -0.793;
   1:  PR[GP1:91,2] = PR[GP1:90,2] + 2.355;
   1:L PR[91] 10mm/sec CNT100;
   1:  PR[GP1:91,1] = PR[GP1:90,1] + -1.602;
   1:  PR[GP1:91,2] = PR[GP1:90,2] + 2.483;
   1:L PR[91] 10mm/sec CNT100;
   1:  PR[GP1:91,1] = PR[GP1:90,1] + -2.199;
   1:  PR[GP1:91,2] = PR[GP1:90,2] + 3.179;
   1:L PR[91] 10mm/sec CNT100;
   1:  PR[GP1:91,1] = PR[GP1:90,1] + -2.674;
   1:  PR[GP1:91,2] = PR[GP1:90,2] + 3.640;
   1:L PR[91] 10mm/sec CNT100;
   1:  PR[GP1:91,1] = PR[GP1:90,1] + -3.076;
   1:  PR[GP1:91,2] = PR[GP1:90,2] + 4.573;
   1:L PR[91] 10mm/sec CNT100;
   1:  PR[GP1:91,1] = PR[GP1:90,1] + -3.238;
   1:  PR[GP1:91,2] = PR[GP1:90,2] + 5.144;
   1:L PR[91] 10mm/sec CNT100;
   1:  PR[GP1:91,1] = PR[GP1:90,1] + -4.337;
   1:  PR[GP1:91,2] = PR[GP1:90,2] + 7.506;
   1:L PR[91] 10mm/sec CNT100;
   1:  PR[GP1:91,1] = PR[GP1:90,1] + -4.813;
   1:  PR[GP1:91,2] = PR[GP1:90,2] + 8.363;
   1:L PR[91] 10mm/sec CNT100;
   1:  PR[GP1:91,1] = PR[GP1:90,1] + -6.108;
   1:  PR[GP1:91,2] = PR[GP1:90,2] + 10.110;
   1:L PR[91] 10mm/sec CNT100;
   1:  PR[GP1:91,1] = PR[GP1:90,1] + -7.106;
   1:  PR[GP1:91,2] = PR[GP1:90,2] + 11.253;
   1:L PR[91] 10mm/sec CNT100;
   1:  PR[GP1:91,1] = PR[GP1:90,1] + -8.372;
   1:  PR[GP1:91,2] = PR[GP1:90,2] + 12.396;
   1:L PR[91] 10mm/sec CNT100;
   1:  PR[GP1:91,1] = PR[GP1:90,1] + -10.003;
   1:  PR[GP1:91,2] = PR[GP1:90,2] + 13.618;
   1:L PR[91] 10mm/sec CNT100;
   1:  PR[GP1:91,1] = PR[GP1:90,1] + -11.086;
   1:  PR[GP1:91,2] = PR[GP1:90,2] + 14.262;
   1:L PR[91] 10mm/sec CNT100;
   1:  PR[GP1:91,1] = PR[GP1:90,1] + -13.369;
   1:  PR[GP1:91,2] = PR[GP1:90,2] + 15.321;
   1:L PR[91] 10mm/sec CNT100;
   1:  PR[GP1:91,1] = PR[GP1:90,1] + -14.175;
   1:  PR[GP1:91,2] = PR[GP1:90,2] + 15.604;
   1:L PR[91] 10mm/sec CNT100;
   1:  PR[GP1:91,1] = PR[GP1:90,1] + -17.037;
   1:  PR[GP1:91,2] = PR[GP1:90,2] + 16.263;
   1:L PR[91] 10mm/sec CNT100;
   1:  PR[GP1:91,1] = PR[GP1:90,1] + -17.528;
   1:  PR[GP1:91,2] = PR[GP1:90,2] + 16.332;
   1:L PR[91] 10mm/sec CNT100;
   1:  PR[GP1:91,1] = PR[GP1:90,1] + -20.818;
   1:  PR[GP1:91,2] = PR[GP1:90,2] + 16.390;
   1:L PR[91] 10mm/sec CNT100;
   1:  PR[GP1:91,1] = PR[GP1:90,1] + -21.009;
   1:  PR[GP1:91,2] = PR[GP1:90,2] + 16.379;
   1:L PR[91] 10mm/sec CNT100;
   1:  PR[GP1:91,1] = PR[GP1:90,1] + -24.484;
   1:  PR[GP1:91,2] = PR[GP1:90,2] + 15.705;
   1:L PR[91] 10mm/sec CNT100;
   1:  PR[GP1:91,1] = PR[GP1:90,1] + -27.715;
   1:  PR[GP1:91,2] = PR[GP1:90,2] + 14.319;
   1:L PR[91] 10mm/sec CNT100;
   1:  PR[GP1:91,1] = PR[GP1:90,1] + -27.771;
   1:  PR[GP1:91,2] = PR[GP1:90,2] + 14.288;
   1:L PR[91] 10mm/sec CNT100;
   1:  PR[GP1:91,1] = PR[GP1:90,1] + -30.526;
   1:  PR[GP1:91,2] = PR[GP1:90,2] + 12.331;
   1:L PR[91] 10mm/sec CNT100;
   1:  PR[GP1:91,1] = PR[GP1:90,1] + -30.660;
   1:  PR[GP1:91,2] = PR[GP1:90,2] + 12.226;
   1:L PR[91] 10mm/sec CNT100;
   1:  PR[GP1:91,1] = PR[GP1:90,1] + -33.029;
   1:  PR[GP1:91,2] = PR[GP1:90,2] + 9.635;
   1:L PR[91] 10mm/sec CNT100;
   1:  PR[GP1:91,1] = PR[GP1:90,1] + -33.160;
   1:  PR[GP1:91,2] = PR[GP1:90,2] + 9.433;
   1:L PR[91] 10mm/sec CNT100;
   1:  PR[GP1:91,1] = PR[GP1:90,1] + -34.790;
   1:  PR[GP1:91,2] = PR[GP1:90,2] + 6.645;
   1:L PR[91] 10mm/sec CNT100;
   1:  PR[GP1:91,1] = PR[GP1:90,1] + -34.901;
   1:  PR[GP1:91,2] = PR[GP1:90,2] + 6.392;
   1:L PR[91] 10mm/sec CNT100;
   1:  PR[GP1:91,1] = PR[GP1:90,1] + -35.902;
   1:  PR[GP1:91,2] = PR[GP1:90,2] + 3.355;
   1:L PR[91] 10mm/sec CNT100;
   1:  PR[GP1:91,1] = PR[GP1:90,1] + -35.970;
   1:  PR[GP1:91,2] = PR[GP1:90,2] + 3.086;
   1:L PR[91] 10mm/sec CNT100;
   1:  PR[GP1:91,1] = PR[GP1:90,1] + -36.327;
   1:  PR[GP1:91,2] = PR[GP1:90,2] + -0.379;
   1:L PR[91] 10mm/sec CNT100;
   1:  PR[GP1:91,1] = PR[GP1:90,1] + -35.957;
   1:  PR[GP1:91,2] = PR[GP1:90,2] + -3.877;
   1:L PR[91] 10mm/sec CNT100;
   1:  PR[GP1:91,1] = PR[GP1:90,1] + -35.912;
   1:  PR[GP1:91,2] = PR[GP1:90,2] + -4.054;
   1:L PR[91] 10mm/sec CNT100;
   1:  PR[GP1:91,1] = PR[GP1:90,1] + -34.855;
   1:  PR[GP1:91,2] = PR[GP1:90,2] + -7.263;
   1:L PR[91] 10mm/sec CNT100;
   1:  PR[GP1:91,1] = PR[GP1:90,1] + -34.822;
   1:  PR[GP1:91,2] = PR[GP1:90,2] + -7.339;
   1:L PR[91] 10mm/sec CNT100;
   1:  PR[GP1:91,1] = PR[GP1:90,1] + -33.033;
   1:  PR[GP1:91,2] = PR[GP1:90,2] + -10.382;
   1:L PR[91] 10mm/sec CNT100;
   1:  PR[GP1:91,1] = PR[GP1:90,1] + -30.604;
   1:  PR[GP1:91,2] = PR[GP1:90,2] + -13.005;
   1:L PR[91] 10mm/sec CNT100;
   1:  PR[GP1:91,1] = PR[GP1:90,1] + -30.474;
   1:  PR[GP1:91,2] = PR[GP1:90,2] + -13.105;
   1:L PR[91] 10mm/sec CNT100;
   1:  PR[GP1:91,1] = PR[GP1:90,1] + -27.714;
   1:  PR[GP1:91,2] = PR[GP1:90,2] + -15.050;
   1:L PR[91] 10mm/sec CNT100;
   1:  PR[GP1:91,1] = PR[GP1:90,1] + -27.285;
   1:  PR[GP1:91,2] = PR[GP1:90,2] + -15.261;
   1:L PR[91] 10mm/sec CNT100;
   1:  PR[GP1:91,1] = PR[GP1:90,1] + -24.505;
   1:  PR[GP1:91,2] = PR[GP1:90,2] + -16.454;
   1:L PR[91] 10mm/sec CNT100;
   1:  PR[GP1:91,1] = PR[GP1:90,1] + -22.897;
   1:  PR[GP1:91,2] = PR[GP1:90,2] + -16.873;
   1:  PR[GP1:91,3] = PR[GP1:90,3] + 12.100;
   1:L PR[91] 10mm/sec CNT100;
   1:  PR[GP1:91,1] = PR[GP1:90,1] + -21.210;
   1:  PR[GP1:91,2] = PR[GP1:90,2] + -17.209;
   1:L PR[91] 10mm/sec CNT100;
   1:  PR[GP1:91,1] = PR[GP1:90,1] + -19.043;
   1:  PR[GP1:91,2] = PR[GP1:90,2] + -17.334;
   1:L PR[91] 10mm/sec CNT100;
   1:  PR[GP1:91,1] = PR[GP1:90,1] + -17.889;
   1:  PR[GP1:91,2] = PR[GP1:90,2] + -17.320;
   1:L PR[91] 10mm/sec CNT100;
   1:  PR[GP1:91,1] = PR[GP1:90,1] + -15.205;
   1:  PR[GP1:91,2] = PR[GP1:90,2] + -16.935;
   1:L PR[91] 10mm/sec CNT100;
   1:  PR[GP1:91,1] = PR[GP1:90,1] + -14.683;
   1:  PR[GP1:91,2] = PR[GP1:90,2] + -16.817;
   1:L PR[91] 10mm/sec CNT100;
   1:  PR[GP1:91,1] = PR[GP1:90,1] + -11.636;
   1:  PR[GP1:91,2] = PR[GP1:90,2] + -15.732;
   1:L PR[91] 10mm/sec CNT100;
   1:  PR[GP1:91,1] = PR[GP1:90,1] + -8.955;
   1:  PR[GP1:91,2] = PR[GP1:90,2] + -14.190;
   1:L PR[91] 10mm/sec CNT100;
   1:  PR[GP1:91,1] = PR[GP1:90,1] + -8.532;
   1:  PR[GP1:91,2] = PR[GP1:90,2] + -13.921;
   1:L PR[91] 10mm/sec CNT100;
   1:  PR[GP1:91,1] = PR[GP1:90,1] + -6.608;
   1:  PR[GP1:91,2] = PR[GP1:90,2] + -12.208;
   1:L PR[91] 10mm/sec CNT100;
   1:  PR[GP1:91,1] = PR[GP1:90,1] + -5.903;
   1:  PR[GP1:91,2] = PR[GP1:90,2] + -11.515;
   1:L PR[91] 10mm/sec CNT100;
   1:  PR[GP1:91,1] = PR[GP1:90,1] + -4.632;
   1:  PR[GP1:91,2] = PR[GP1:90,2] + -9.784;
   1:L PR[91] 10mm/sec CNT100;
   1:  PR[GP1:91,1] = PR[GP1:90,1] + -3.893;
   1:  PR[GP1:91,2] = PR[GP1:90,2] + -8.661;
   1:L PR[91] 10mm/sec CNT100;
   1:  PR[GP1:91,1] = PR[GP1:90,1] + -3.127;
   1:  PR[GP1:91,2] = PR[GP1:90,2] + -6.990;
   1:L PR[91] 10mm/sec CNT100;
   1:  PR[GP1:91,1] = PR[GP1:90,1] + -2.738;
   1:  PR[GP1:91,2] = PR[GP1:90,2] + -6.377;
   1:L PR[91] 10mm/sec CNT100;
   1:  PR[GP1:91,1] = PR[GP1:90,1] + -2.529;
   1:  PR[GP1:91,2] = PR[GP1:90,2] + -5.992;
   1:L PR[91] 10mm/sec CNT100;
   1:  PR[GP1:91,1] = PR[GP1:90,1] + -1.810;
   1:  PR[GP1:91,2] = PR[GP1:90,2] + -5.426;
   1:L PR[91] 10mm/sec CNT100;
   1:  PR[GP1:91,1] = PR[GP1:90,1] + -1.561;
   1:  PR[GP1:91,2] = PR[GP1:90,2] + -5.162;
   1:L PR[91] 10mm/sec CNT100;
   1:  PR[GP1:91,1] = PR[GP1:90,1] + -0.661;
   1:  PR[GP1:91,2] = PR[GP1:90,2] + -5.075;
   1:L PR[91] 10mm/sec CNT100;
   1:  PR[GP1:91,1] = PR[GP1:90,1] + -0.253;
   1:  PR[GP1:91,2] = PR[GP1:90,2] + -5.004;
   1:L PR[91] 10mm/sec CNT100;
   1:  PR[GP1:91,1] = PR[GP1:90,1] + 0.863;
   1:  PR[GP1:91,2] = PR[GP1:90,2] + -5.725;
   1:L PR[91] 10mm/sec CNT100;
   1:  PR[GP1:91,1] = PR[GP1:90,1] + 1.471;
   1:  PR[GP1:91,2] = PR[GP1:90,2] + -6.799;
   1:L PR[91] 10mm/sec CNT100;
   1:  PR[GP1:91,1] = PR[GP1:90,1] + 2.673;
   1:  PR[GP1:91,2] = PR[GP1:90,2] + -9.167;
   1:L PR[91] 10mm/sec CNT100;
   1:  PR[GP1:91,1] = PR[GP1:90,1] + 4.213;
   1:  PR[GP1:91,2] = PR[GP1:90,2] + -11.260;
   1:L PR[91] 10mm/sec CNT100;
   1:  PR[GP1:91,1] = PR[GP1:90,1] + 4.669;
   1:  PR[GP1:91,2] = PR[GP1:90,2] + -11.731;
   1:L PR[91] 10mm/sec CNT100;
   1:  PR[GP1:91,1] = PR[GP1:90,1] + 6.068;
   1:  PR[GP1:91,2] = PR[GP1:90,2] + -13.085;
   1:L PR[91] 10mm/sec CNT100;
   1:  PR[GP1:91,1] = PR[GP1:90,1] + 7.160;
   1:  PR[GP1:91,2] = PR[GP1:90,2] + -13.894;
   1:L PR[91] 10mm/sec CNT100;
   1:  PR[GP1:91,1] = PR[GP1:90,1] + 8.202;
   1:  PR[GP1:91,2] = PR[GP1:90,2] + -14.622;
   1:L PR[91] 10mm/sec CNT100;
   1:  PR[GP1:91,1] = PR[GP1:90,1] + 10.585;
   1:  PR[GP1:91,2] = PR[GP1:90,2] + -15.848;
   1:L PR[91] 10mm/sec CNT100;
   1:  PR[GP1:91,1] = PR[GP1:90,1] + 11.525;
   1:  PR[GP1:91,2] = PR[GP1:90,2] + -16.164;
   1:L PR[91] 10mm/sec CNT100;
   1:  PR[GP1:91,1] = PR[GP1:90,1] + 13.242;
   1:  PR[GP1:91,2] = PR[GP1:90,2] + -16.771;
   1:L PR[91] 10mm/sec CNT100;
   1:  PR[GP1:91,1] = PR[GP1:90,1] + 16.065;
   1:  PR[GP1:91,2] = PR[GP1:90,2] + -17.311;
   1:L PR[91] 10mm/sec CNT100;
   1:  PR[GP1:91,1] = PR[GP1:90,1] + 18.937;
   1:  PR[GP1:91,2] = PR[GP1:90,2] + -17.430;
   1:L PR[91] 10mm/sec CNT100;
   1:  PR[GP1:91,1] = PR[GP1:90,1] + 21.710;
   1:  PR[GP1:91,2] = PR[GP1:90,2] + -17.153;
   1:L PR[91] 10mm/sec CNT100;
   1:  PR[GP1:91,1] = PR[GP1:90,1] + 24.399;
   1:  PR[GP1:91,2] = PR[GP1:90,2] + -16.470;
   1:L PR[91] 10mm/sec CNT100;
   1:  PR[GP1:91,1] = PR[GP1:90,1] + 26.944;
   1:  PR[GP1:91,2] = PR[GP1:90,2] + -15.401;
   1:L PR[91] 10mm/sec CNT100;
   1:  PR[GP1:91,1] = PR[GP1:90,1] + 28.399;
   1:  PR[GP1:91,2] = PR[GP1:90,2] + -14.513;
   1:L PR[91] 10mm/sec CNT100;
   1:  PR[GP1:91,1] = PR[GP1:90,1] + 29.256;
   1:  PR[GP1:91,2] = PR[GP1:90,2] + -13.981;
   1:L PR[91] 10mm/sec CNT100;
   1:  PR[GP1:91,1] = PR[GP1:90,1] + 31.279;
   1:  PR[GP1:91,2] = PR[GP1:90,2] + -12.243;
   1:L PR[91] 10mm/sec CNT100;
   1:  PR[GP1:91,1] = PR[GP1:90,1] + 33.003;
   1:  PR[GP1:91,2] = PR[GP1:90,2] + -10.220;
   1:L PR[91] 10mm/sec CNT100;
   1:  PR[GP1:91,1] = PR[GP1:90,1] + 34.389;
   1:  PR[GP1:91,2] = PR[GP1:90,2] + -7.960;
   1:L PR[91] 10mm/sec CNT100;
   1:  PR[GP1:91,1] = PR[GP1:90,1] + 35.403;
   1:  PR[GP1:91,2] = PR[GP1:90,2] + -5.519;
   1:L PR[91] 10mm/sec CNT100;
   1:  PR[GP1:91,1] = PR[GP1:90,1] + 36.021;
   1:  PR[GP1:91,2] = PR[GP1:90,2] + -2.955;
   1:L PR[91] 10mm/sec CNT100;
   1:  PR[GP1:91,1] = PR[GP1:90,1] + 36.126;
   1:  PR[GP1:91,2] = PR[GP1:90,2] + -1.647;
   1:L PR[91] 10mm/sec CNT100;
   1:  PR[GP1:91,1] = PR[GP1:90,1] + 36.271;
   1:  PR[GP1:91,2] = PR[GP1:90,2] + -0.328;
   1:L PR[91] 10mm/sec CNT100;
   1:  PR[GP1:91,1] = PR[GP1:90,1] + 36.052;
   1:  PR[GP1:91,2] = PR[GP1:90,2] + 1.533;
   1:L PR[91] 10mm/sec CNT100;
   1:  PR[GP1:91,1] = PR[GP1:90,1] + 35.900;
   1:  PR[GP1:91,2] = PR[GP1:90,2] + 2.981;
   1:L PR[91] 10mm/sec CNT100;
   1:  PR[GP1:91,1] = PR[GP1:90,1] + 34.909;
   1:  PR[GP1:91,2] = PR[GP1:90,2] + 6.164;
   1:L PR[91] 10mm/sec CNT100;
   1:  PR[GP1:91,1] = PR[GP1:90,1] + 33.304;
   1:  PR[GP1:91,2] = PR[GP1:90,2] + 9.092;
   1:L PR[91] 10mm/sec CNT100;
   1:  PR[GP1:91,1] = PR[GP1:90,1] + 31.145;
   1:  PR[GP1:91,2] = PR[GP1:90,2] + 11.650;
   1:L PR[91] 10mm/sec CNT100;
   1:  PR[GP1:91,1] = PR[GP1:90,1] + 28.518;
   1:  PR[GP1:91,2] = PR[GP1:90,2] + 13.739;
   1:L PR[91] 10mm/sec CNT100;
   1:  PR[GP1:91,1] = PR[GP1:90,1] + 26.446;
   1:  PR[GP1:91,2] = PR[GP1:90,2] + 14.804;
   1:L PR[91] 10mm/sec CNT100;
   1:  PR[GP1:91,1] = PR[GP1:90,1] + 25.507;
   1:  PR[GP1:91,2] = PR[GP1:90,2] + 15.272;
   1:L PR[91] 10mm/sec CNT100;
   1:  PR[GP1:91,1] = PR[GP1:90,1] + 22.176;
   1:  PR[GP1:91,2] = PR[GP1:90,2] + 16.193;
   1:L PR[91] 10mm/sec CNT100;
   1:  PR[GP1:91,1] = PR[GP1:90,1] + 18.714;
   1:  PR[GP1:91,2] = PR[GP1:90,2] + 16.464;
   1:L PR[91] 10mm/sec CNT100;
   1:  PR[GP1:91,1] = PR[GP1:90,1] + 15.242;
   1:  PR[GP1:91,2] = PR[GP1:90,2] + 16.073;
   1:L PR[91] 10mm/sec CNT100;
   1:  PR[GP1:91,1] = PR[GP1:90,1] + 11.829;
   1:  PR[GP1:91,2] = PR[GP1:90,2] + 15.026;
   1:L PR[91] 10mm/sec CNT100;
   1:  PR[GP1:91,1] = PR[GP1:90,1] + 8.660;
   1:  PR[GP1:91,2] = PR[GP1:90,2] + 13.370;
   1:L PR[91] 10mm/sec CNT100;
   1:  PR[GP1:91,1] = PR[GP1:90,1] + 5.856;
   1:  PR[GP1:91,2] = PR[GP1:90,2] + 11.170;
   1:L PR[91] 10mm/sec CNT100;
   1:  PR[GP1:91,1] = PR[GP1:90,1] + 3.529;
   1:  PR[GP1:91,2] = PR[GP1:90,2] + 8.503;
   1:L PR[91] 10mm/sec CNT100;
   1:  PR[GP1:91,1] = PR[GP1:90,1] + 1.799;
   1:  PR[GP1:91,2] = PR[GP1:90,2] + 5.499;
   1:L PR[91] 10mm/sec CNT100;
   1:  PR[GP1:91,1] = PR[GP1:90,1] + 1.655;
   1:  PR[GP1:91,2] = PR[GP1:90,2] + 5.064;
   1:L PR[91] 10mm/sec CNT100;
   1:  PR[GP1:91,1] = PR[GP1:90,1] + 1.519;
   1:  PR[GP1:91,2] = PR[GP1:90,2] + 4.815;
   1:L PR[91] 10mm/sec CNT100;
   1:  PR[GP1:91,1] = PR[GP1:90,1] + 0.891;
   1:  PR[GP1:91,2] = PR[GP1:90,2] + 3.884;
   1:L PR[91] 10mm/sec CNT100;
   1:  PR[GP1:91,1] = PR[GP1:90,1] + 0.445;
   1:  PR[GP1:91,2] = PR[GP1:90,2] + 3.624;
   1:L PR[91] 10mm/sec CNT100;
   1:  PR[GP1:91,1] = PR[GP1:90,1] + -0.467;
   1:  PR[GP1:91,2] = PR[GP1:90,2] + 3.265;
   1:L PR[91] 10mm/sec CNT100;
   1:  PR[GP1:91,1] = PR[GP1:90,1] + -1.486;
   1:  PR[GP1:91,2] = PR[GP1:90,2] + 3.656;
   1:L PR[91] 10mm/sec CNT100;
   1:  PR[GP1:91,1] = PR[GP1:90,1] + -1.814;
   1:  PR[GP1:91,2] = PR[GP1:90,2] + 3.708;
   1:L PR[91] 10mm/sec CNT100;
   1:  PR[GP1:91,1] = PR[GP1:90,1] + -2.404;
   1:  PR[GP1:91,2] = PR[GP1:90,2] + 4.396;
   1:L PR[91] 10mm/sec CNT100;
   1:  PR[GP1:91,1] = PR[GP1:90,1] + -2.828;
   1:  PR[GP1:91,2] = PR[GP1:90,2] + 4.810;
   1:L PR[91] 10mm/sec CNT100;
   1:  PR[GP1:91,1] = PR[GP1:90,1] + -4.413;
   1:  PR[GP1:91,2] = PR[GP1:90,2] + 8.005;
   1:L PR[91] 10mm/sec CNT100;
   1:  PR[GP1:91,1] = PR[GP1:90,1] + -6.275;
   1:  PR[GP1:91,2] = PR[GP1:90,2] + 10.514;
   1:L PR[91] 10mm/sec CNT100;
   1:  PR[GP1:91,1] = PR[GP1:90,1] + -6.622;
   1:  PR[GP1:91,2] = PR[GP1:90,2] + 10.911;
   1:L PR[91] 10mm/sec CNT100;
   1:  PR[GP1:91,1] = PR[GP1:90,1] + -8.557;
   1:  PR[GP1:91,2] = PR[GP1:90,2] + 12.658;
   1:L PR[91] 10mm/sec CNT100;
   1:  PR[GP1:91,1] = PR[GP1:90,1] + -9.454;
   1:  PR[GP1:91,2] = PR[GP1:90,2] + 13.330;
   1:L PR[91] 10mm/sec CNT100;
   1:  PR[GP1:91,1] = PR[GP1:90,1] + -11.258;
   1:  PR[GP1:91,2] = PR[GP1:90,2] + 14.402;
   1:L PR[91] 10mm/sec CNT100;
   1:  PR[GP1:91,1] = PR[GP1:90,1] + -12.771;
   1:  PR[GP1:91,2] = PR[GP1:90,2] + 15.104;
   1:L PR[91] 10mm/sec CNT100;
   1:  PR[GP1:91,1] = PR[GP1:90,1] + -14.314;
   1:  PR[GP1:91,2] = PR[GP1:90,2] + 15.647;
   1:L PR[91] 10mm/sec CNT100;
   1:  PR[GP1:91,1] = PR[GP1:90,1] + -16.408;
   1:  PR[GP1:91,2] = PR[GP1:90,2] + 16.128;
   1:L PR[91] 10mm/sec CNT100;
   1:  PR[GP1:91,1] = PR[GP1:90,1] + -17.622;
   1:  PR[GP1:91,2] = PR[GP1:90,2] + 16.299;
   1:L PR[91] 10mm/sec CNT100;
   1:  PR[GP1:91,1] = PR[GP1:90,1] + -20.177;
   1:  PR[GP1:91,2] = PR[GP1:90,2] + 16.345;
   1:L PR[91] 10mm/sec CNT100;
   1:  PR[GP1:91,1] = PR[GP1:90,1] + -21.052;
   1:  PR[GP1:91,2] = PR[GP1:90,2] + 16.293;
   1:L PR[91] 10mm/sec CNT100;
   1:  PR[GP1:91,1] = PR[GP1:90,1] + -23.885;
   1:  PR[GP1:91,2] = PR[GP1:90,2] + 15.745;
   1:L PR[91] 10mm/sec CNT100;
   1:  PR[GP1:91,1] = PR[GP1:90,1] + -24.455;
   1:  PR[GP1:91,2] = PR[GP1:90,2] + 15.594;
   1:L PR[91] 10mm/sec CNT100;
   1:  PR[GP1:91,1] = PR[GP1:90,1] + -27.347;
   1:  PR[GP1:91,2] = PR[GP1:90,2] + 14.368;
   1:L PR[91] 10mm/sec CNT100;
   1:  PR[GP1:91,1] = PR[GP1:90,1] + -27.675;
   1:  PR[GP1:91,2] = PR[GP1:90,2] + 14.206;
   1:L PR[91] 10mm/sec CNT100;
   1:  PR[GP1:91,1] = PR[GP1:90,1] + -30.397;
   1:  PR[GP1:91,2] = PR[GP1:90,2] + 12.294;
   1:L PR[91] 10mm/sec CNT100;
   1:  PR[GP1:91,1] = PR[GP1:90,1] + -30.555;
   1:  PR[GP1:91,2] = PR[GP1:90,2] + 12.171;
   1:L PR[91] 10mm/sec CNT100;
   1:  PR[GP1:91,1] = PR[GP1:90,1] + -32.961;
   1:  PR[GP1:91,2] = PR[GP1:90,2] + 9.557;
   1:L PR[91] 10mm/sec CNT100;
   1:  PR[GP1:91,1] = PR[GP1:90,1] + -34.756;
   1:  PR[GP1:91,2] = PR[GP1:90,2] + 6.499;
   1:L PR[91] 10mm/sec CNT100;
   1:  PR[GP1:91,1] = PR[GP1:90,1] + -35.868;
   1:  PR[GP1:91,2] = PR[GP1:90,2] + 3.126;
   1:L PR[91] 10mm/sec CNT100;
   1:  PR[GP1:91,1] = PR[GP1:90,1] + -36.237;
   1:  PR[GP1:91,2] = PR[GP1:90,2] + -0.408;
   1:L PR[91] 10mm/sec CNT100;
   1:  PR[GP1:91,1] = PR[GP1:90,1] + -35.891;
   1:  PR[GP1:91,2] = PR[GP1:90,2] + -3.515;
   1:L PR[91] 10mm/sec CNT100;
   1:  PR[GP1:91,1] = PR[GP1:90,1] + -35.831;
   1:  PR[GP1:91,2] = PR[GP1:90,2] + -3.946;
   1:L PR[91] 10mm/sec CNT100;
   1:  PR[GP1:91,1] = PR[GP1:90,1] + -35.771;
   1:  PR[GP1:91,2] = PR[GP1:90,2] + -4.133;
   1:L PR[91] 10mm/sec CNT100;
   1:  PR[GP1:91,1] = PR[GP1:90,1] + -34.702;
   1:  PR[GP1:91,2] = PR[GP1:90,2] + -7.318;
   1:L PR[91] 10mm/sec CNT100;
   1:  PR[GP1:91,1] = PR[GP1:90,1] + -32.891;
   1:  PR[GP1:91,2] = PR[GP1:90,2] + -10.380;
   1:L PR[91] 10mm/sec CNT100;
   1:  PR[GP1:91,1] = PR[GP1:90,1] + -32.511;
   1:  PR[GP1:91,2] = PR[GP1:90,2] + -10.817;
   1:L PR[91] 10mm/sec CNT100;
   1:  PR[GP1:91,1] = PR[GP1:90,1] + -30.505;
   1:  PR[GP1:91,2] = PR[GP1:90,2] + -12.982;
   1:L PR[91] 10mm/sec CNT100;
   1:  PR[GP1:91,1] = PR[GP1:90,1] + -29.811;
   1:  PR[GP1:91,2] = PR[GP1:90,2] + -13.516;
   1:L PR[91] 10mm/sec CNT100;
   1:  PR[GP1:91,1] = PR[GP1:90,1] + -27.667;
   1:  PR[GP1:91,2] = PR[GP1:90,2] + -15.028;
   1:L PR[91] 10mm/sec CNT100;
   1:  PR[GP1:91,1] = PR[GP1:90,1] + -26.552;
   1:  PR[GP1:91,2] = PR[GP1:90,2] + -15.575;
   1:L PR[91] 10mm/sec CNT100;
   1:  PR[GP1:91,1] = PR[GP1:90,1] + -24.518;
   1:  PR[GP1:91,2] = PR[GP1:90,2] + -16.447;
   1:L PR[91] 10mm/sec CNT100;
   1:  PR[GP1:91,1] = PR[GP1:90,1] + -22.116;
   1:  PR[GP1:91,2] = PR[GP1:90,2] + -17.075;
   1:  PR[GP1:91,3] = PR[GP1:90,3] + 13.200;
   1:L PR[91] 10mm/sec CNT100;
   1:  PR[GP1:91,1] = PR[GP1:90,1] + -21.289;
   1:  PR[GP1:91,2] = PR[GP1:90,2] + -17.240;
   1:L PR[91] 10mm/sec CNT100;
   1:  PR[GP1:91,1] = PR[GP1:90,1] + -18.238;
   1:  PR[GP1:91,2] = PR[GP1:90,2] + -17.415;
   1:L PR[91] 10mm/sec CNT100;
   1:  PR[GP1:91,1] = PR[GP1:90,1] + -18.034;
   1:  PR[GP1:91,2] = PR[GP1:90,2] + -17.413;
   1:L PR[91] 10mm/sec CNT100;
   1:  PR[GP1:91,1] = PR[GP1:90,1] + -16.724;
   1:  PR[GP1:91,2] = PR[GP1:90,2] + -17.225;
   1:L PR[91] 10mm/sec CNT100;
   1:  PR[GP1:91,1] = PR[GP1:90,1] + -14.857;
   1:  PR[GP1:91,2] = PR[GP1:90,2] + -16.992;
   1:L PR[91] 10mm/sec CNT100;
   1:  PR[GP1:91,1] = PR[GP1:90,1] + -14.566;
   1:  PR[GP1:91,2] = PR[GP1:90,2] + -16.945;
   1:L PR[91] 10mm/sec CNT100;
   1:  PR[GP1:91,1] = PR[GP1:90,1] + -11.971;
   1:  PR[GP1:91,2] = PR[GP1:90,2] + -16.081;
   1:L PR[91] 10mm/sec CNT100;
   1:  PR[GP1:91,1] = PR[GP1:90,1] + -11.113;
   1:  PR[GP1:91,2] = PR[GP1:90,2] + -15.756;
   1:L PR[91] 10mm/sec CNT100;
   1:  PR[GP1:91,1] = PR[GP1:90,1] + -9.298;
   1:  PR[GP1:91,2] = PR[GP1:90,2] + -14.712;
   1:L PR[91] 10mm/sec CNT100;
   1:  PR[GP1:91,1] = PR[GP1:90,1] + -7.994;
   1:  PR[GP1:91,2] = PR[GP1:90,2] + -13.883;
   1:L PR[91] 10mm/sec CNT100;
   1:  PR[GP1:91,1] = PR[GP1:90,1] + -6.891;
   1:  PR[GP1:91,2] = PR[GP1:90,2] + -12.901;
   1:L PR[91] 10mm/sec CNT100;
   1:  PR[GP1:91,1] = PR[GP1:90,1] + -5.376;
   1:  PR[GP1:91,2] = PR[GP1:90,2] + -11.413;
   1:L PR[91] 10mm/sec CNT100;
   1:  PR[GP1:91,1] = PR[GP1:90,1] + -4.810;
   1:  PR[GP1:91,2] = PR[GP1:90,2] + -10.641;
   1:L PR[91] 10mm/sec CNT100;
   1:  PR[GP1:91,1] = PR[GP1:90,1] + -3.408;
   1:  PR[GP1:91,2] = PR[GP1:90,2] + -8.514;
   1:L PR[91] 10mm/sec CNT100;
   1:  PR[GP1:91,1] = PR[GP1:90,1] + -3.136;
   1:  PR[GP1:91,2] = PR[GP1:90,2] + -7.921;
   1:L PR[91] 10mm/sec CNT100;
   1:  PR[GP1:91,1] = PR[GP1:90,1] + -2.676;
   1:  PR[GP1:91,2] = PR[GP1:90,2] + -7.200;
   1:L PR[91] 10mm/sec CNT100;
   1:  PR[GP1:91,1] = PR[GP1:90,1] + -2.388;
   1:  PR[GP1:91,2] = PR[GP1:90,2] + -6.901;
   1:L PR[91] 10mm/sec CNT100;
   1:  PR[GP1:91,1] = PR[GP1:90,1] + -1.666;
   1:  PR[GP1:91,2] = PR[GP1:90,2] + -6.418;
   1:L PR[91] 10mm/sec CNT100;
   1:  PR[GP1:91,1] = PR[GP1:90,1] + -1.340;
   1:  PR[GP1:91,2] = PR[GP1:90,2] + -6.320;
   1:L PR[91] 10mm/sec CNT100;
   1:  PR[GP1:91,1] = PR[GP1:90,1] + -0.462;
   1:  PR[GP1:91,2] = PR[GP1:90,2] + -6.263;
   1:L PR[91] 10mm/sec CNT100;
   1:  PR[GP1:91,1] = PR[GP1:90,1] + -0.142;
   1:  PR[GP1:91,2] = PR[GP1:90,2] + -6.363;
   1:L PR[91] 10mm/sec CNT100;
   1:  PR[GP1:91,1] = PR[GP1:90,1] + 0.633;
   1:  PR[GP1:91,2] = PR[GP1:90,2] + -6.776;
   1:L PR[91] 10mm/sec CNT100;
   1:  PR[GP1:91,1] = PR[GP1:90,1] + 0.912;
   1:  PR[GP1:91,2] = PR[GP1:90,2] + -7.083;
   1:L PR[91] 10mm/sec CNT100;
   1:  PR[GP1:91,1] = PR[GP1:90,1] + 1.331;
   1:  PR[GP1:91,2] = PR[GP1:90,2] + -7.808;
   1:L PR[91] 10mm/sec CNT100;
   1:  PR[GP1:91,1] = PR[GP1:90,1] + 2.201;
   1:  PR[GP1:91,2] = PR[GP1:90,2] + -9.381;
   1:L PR[91] 10mm/sec CNT100;
   1:  PR[GP1:91,1] = PR[GP1:90,1] + 3.681;
   1:  PR[GP1:91,2] = PR[GP1:90,2] + -11.369;
   1:L PR[91] 10mm/sec CNT100;
   1:  PR[GP1:91,1] = PR[GP1:90,1] + 3.833;
   1:  PR[GP1:91,2] = PR[GP1:90,2] + -11.551;
   1:L PR[91] 10mm/sec CNT100;
   1:  PR[GP1:91,1] = PR[GP1:90,1] + 5.715;
   1:  PR[GP1:91,2] = PR[GP1:90,2] + -13.353;
   1:L PR[91] 10mm/sec CNT100;
   1:  PR[GP1:91,1] = PR[GP1:90,1] + 7.875;
   1:  PR[GP1:91,2] = PR[GP1:90,2] + -14.866;
   1:L PR[91] 10mm/sec CNT100;
   1:  PR[GP1:91,1] = PR[GP1:90,1] + 8.770;
   1:  PR[GP1:91,2] = PR[GP1:90,2] + -15.331;
   1:L PR[91] 10mm/sec CNT100;
   1:  PR[GP1:91,1] = PR[GP1:90,1] + 10.257;
   1:  PR[GP1:91,2] = PR[GP1:90,2] + -16.056;
   1:L PR[91] 10mm/sec CNT100;
   1:  PR[GP1:91,1] = PR[GP1:90,1] + 12.284;
   1:  PR[GP1:91,2] = PR[GP1:90,2] + -16.738;
   1:L PR[91] 10mm/sec CNT100;
   1:  PR[GP1:91,1] = PR[GP1:90,1] + 12.827;
   1:  PR[GP1:91,2] = PR[GP1:90,2] + -16.908;
   1:L PR[91] 10mm/sec CNT100;
   1:  PR[GP1:91,1] = PR[GP1:90,1] + 14.160;
   1:  PR[GP1:91,2] = PR[GP1:90,2] + -17.143;
   1:L PR[91] 10mm/sec CNT100;
   1:  PR[GP1:91,1] = PR[GP1:90,1] + 15.613;
   1:  PR[GP1:91,2] = PR[GP1:90,2] + -17.421;
   1:L PR[91] 10mm/sec CNT100;
   1:  PR[GP1:91,1] = PR[GP1:90,1] + 18.503;
   1:  PR[GP1:91,2] = PR[GP1:90,2] + -17.538;
   1:L PR[91] 10mm/sec CNT100;
   1:  PR[GP1:91,1] = PR[GP1:90,1] + 21.375;
   1:  PR[GP1:91,2] = PR[GP1:90,2] + -17.234;
   1:L PR[91] 10mm/sec CNT100;
   1:  PR[GP1:91,1] = PR[GP1:90,1] + 24.080;
   1:  PR[GP1:91,2] = PR[GP1:90,2] + -16.544;
   1:L PR[91] 10mm/sec CNT100;
   1:  PR[GP1:91,1] = PR[GP1:90,1] + 26.631;
   1:  PR[GP1:91,2] = PR[GP1:90,2] + -15.469;
   1:L PR[91] 10mm/sec CNT100;
   1:  PR[GP1:91,1] = PR[GP1:90,1] + 28.976;
   1:  PR[GP1:91,2] = PR[GP1:90,2] + -14.035;
   1:L PR[91] 10mm/sec CNT100;
   1:  PR[GP1:91,1] = PR[GP1:90,1] + 31.060;
   1:  PR[GP1:91,2] = PR[GP1:90,2] + -12.278;
   1:L PR[91] 10mm/sec CNT100;
   1:  PR[GP1:91,1] = PR[GP1:90,1] + 32.812;
   1:  PR[GP1:91,2] = PR[GP1:90,2] + -10.247;
   1:L PR[91] 10mm/sec CNT100;
   1:  PR[GP1:91,1] = PR[GP1:90,1] + 34.195;
   1:  PR[GP1:91,2] = PR[GP1:90,2] + -7.986;
   1:L PR[91] 10mm/sec CNT100;
   1:  PR[GP1:91,1] = PR[GP1:90,1] + 35.208;
   1:  PR[GP1:91,2] = PR[GP1:90,2] + -5.543;
   1:L PR[91] 10mm/sec CNT100;
   1:  PR[GP1:91,1] = PR[GP1:90,1] + 35.824;
   1:  PR[GP1:91,2] = PR[GP1:90,2] + -2.976;
   1:L PR[91] 10mm/sec CNT100;
   1:  PR[GP1:91,1] = PR[GP1:90,1] + 35.879;
   1:  PR[GP1:91,2] = PR[GP1:90,2] + -2.293;
   1:L PR[91] 10mm/sec CNT100;
   1:  PR[GP1:91,1] = PR[GP1:90,1] + 36.055;
   1:  PR[GP1:91,2] = PR[GP1:90,2] + -0.702;
   1:L PR[91] 10mm/sec CNT100;
   1:  PR[GP1:91,1] = PR[GP1:90,1] + 36.082;
   1:  PR[GP1:91,2] = PR[GP1:90,2] + -0.355;
   1:L PR[91] 10mm/sec CNT100;
   1:  PR[GP1:91,1] = PR[GP1:90,1] + 35.712;
   1:  PR[GP1:91,2] = PR[GP1:90,2] + 2.962;
   1:L PR[91] 10mm/sec CNT100;
   1:  PR[GP1:91,1] = PR[GP1:90,1] + 34.718;
   1:  PR[GP1:91,2] = PR[GP1:90,2] + 6.149;
   1:L PR[91] 10mm/sec CNT100;
   1:  PR[GP1:91,1] = PR[GP1:90,1] + 33.109;
   1:  PR[GP1:91,2] = PR[GP1:90,2] + 9.076;
   1:L PR[91] 10mm/sec CNT100;
   1:  PR[GP1:91,1] = PR[GP1:90,1] + 30.950;
   1:  PR[GP1:91,2] = PR[GP1:90,2] + 11.631;
   1:L PR[91] 10mm/sec CNT100;
   1:  PR[GP1:91,1] = PR[GP1:90,1] + 28.261;
   1:  PR[GP1:91,2] = PR[GP1:90,2] + 13.713;
   1:L PR[91] 10mm/sec CNT100;
   1:  PR[GP1:91,1] = PR[GP1:90,1] + 25.188;
   1:  PR[GP1:91,2] = PR[GP1:90,2] + 15.245;
   1:L PR[91] 10mm/sec CNT100;
   1:  PR[GP1:91,1] = PR[GP1:90,1] + 21.862;
   1:  PR[GP1:91,2] = PR[GP1:90,2] + 16.164;
   1:L PR[91] 10mm/sec CNT100;
   1:  PR[GP1:91,1] = PR[GP1:90,1] + 18.386;
   1:  PR[GP1:91,2] = PR[GP1:90,2] + 16.432;
   1:L PR[91] 10mm/sec CNT100;
   1:  PR[GP1:91,1] = PR[GP1:90,1] + 14.826;
   1:  PR[GP1:91,2] = PR[GP1:90,2] + 16.029;
   1:L PR[91] 10mm/sec CNT100;
   1:  PR[GP1:91,1] = PR[GP1:90,1] + 11.399;
   1:  PR[GP1:91,2] = PR[GP1:90,2] + 14.978;
   1:L PR[91] 10mm/sec CNT100;
   1:  PR[GP1:91,1] = PR[GP1:90,1] + 8.181;
   1:  PR[GP1:91,2] = PR[GP1:90,2] + 13.309;
   1:L PR[91] 10mm/sec CNT100;
   1:  PR[GP1:91,1] = PR[GP1:90,1] + 5.350;
   1:  PR[GP1:91,2] = PR[GP1:90,2] + 11.095;
   1:L PR[91] 10mm/sec CNT100;
   1:  PR[GP1:91,1] = PR[GP1:90,1] + 3.016;
   1:  PR[GP1:91,2] = PR[GP1:90,2] + 8.428;
   1:L PR[91] 10mm/sec CNT100;
   1:  PR[GP1:91,1] = PR[GP1:90,1] + 1.469;
   1:  PR[GP1:91,2] = PR[GP1:90,2] + 5.774;
   1:L PR[91] 10mm/sec CNT100;
   1:  PR[GP1:91,1] = PR[GP1:90,1] + 0.643;
   1:  PR[GP1:91,2] = PR[GP1:90,2] + 4.795;
   1:L PR[91] 10mm/sec CNT100;
   1:  PR[GP1:91,1] = PR[GP1:90,1] + -0.634;
   1:  PR[GP1:91,2] = PR[GP1:90,2] + 4.365;
   1:L PR[91] 10mm/sec CNT100;
   1:  PR[GP1:91,1] = PR[GP1:90,1] + -1.987;
   1:  PR[GP1:91,2] = PR[GP1:90,2] + 4.673;
   1:L PR[91] 10mm/sec CNT100;
   1:  PR[GP1:91,1] = PR[GP1:90,1] + -2.362;
   1:  PR[GP1:91,2] = PR[GP1:90,2] + 5.111;
   1:L PR[91] 10mm/sec CNT100;
   1:  PR[GP1:91,1] = PR[GP1:90,1] + -2.941;
   1:  PR[GP1:91,2] = PR[GP1:90,2] + 5.677;
   1:L PR[91] 10mm/sec CNT100;
   1:  PR[GP1:91,1] = PR[GP1:90,1] + -4.002;
   1:  PR[GP1:91,2] = PR[GP1:90,2] + 7.800;
   1:L PR[91] 10mm/sec CNT100;
   1:  PR[GP1:91,1] = PR[GP1:90,1] + -4.525;
   1:  PR[GP1:91,2] = PR[GP1:90,2] + 8.511;
   1:L PR[91] 10mm/sec CNT100;
   1:  PR[GP1:91,1] = PR[GP1:90,1] + -6.178;
   1:  PR[GP1:91,2] = PR[GP1:90,2] + 10.646;
   1:L PR[91] 10mm/sec CNT100;
   1:  PR[GP1:91,1] = PR[GP1:90,1] + -7.753;
   1:  PR[GP1:91,2] = PR[GP1:90,2] + 12.027;
   1:L PR[91] 10mm/sec CNT100;
   1:  PR[GP1:91,1] = PR[GP1:90,1] + -8.741;
   1:  PR[GP1:91,2] = PR[GP1:90,2] + 12.920;
   1:L PR[91] 10mm/sec CNT100;
   1:  PR[GP1:91,1] = PR[GP1:90,1] + -8.905;
   1:  PR[GP1:91,2] = PR[GP1:90,2] + 13.042;
   1:L PR[91] 10mm/sec CNT100;
   1:  PR[GP1:91,1] = PR[GP1:90,1] + -11.430;
   1:  PR[GP1:91,2] = PR[GP1:90,2] + 14.543;
   1:L PR[91] 10mm/sec CNT100;
   1:  PR[GP1:91,1] = PR[GP1:90,1] + -12.173;
   1:  PR[GP1:91,2] = PR[GP1:90,2] + 14.887;
   1:L PR[91] 10mm/sec CNT100;
   1:  PR[GP1:91,1] = PR[GP1:90,1] + -14.453;
   1:  PR[GP1:91,2] = PR[GP1:90,2] + 15.689;
   1:L PR[91] 10mm/sec CNT100;
   1:  PR[GP1:91,1] = PR[GP1:90,1] + -15.779;
   1:  PR[GP1:91,2] = PR[GP1:90,2] + 15.994;
   1:L PR[91] 10mm/sec CNT100;
   1:  PR[GP1:91,1] = PR[GP1:90,1] + -17.716;
   1:  PR[GP1:91,2] = PR[GP1:90,2] + 16.267;
   1:L PR[91] 10mm/sec CNT100;
   1:  PR[GP1:91,1] = PR[GP1:90,1] + -19.537;
   1:  PR[GP1:91,2] = PR[GP1:90,2] + 16.299;
   1:L PR[91] 10mm/sec CNT100;
   1:  PR[GP1:91,1] = PR[GP1:90,1] + -21.095;
   1:  PR[GP1:91,2] = PR[GP1:90,2] + 16.208;
   1:L PR[91] 10mm/sec CNT100;
   1:  PR[GP1:91,1] = PR[GP1:90,1] + -23.253;
   1:  PR[GP1:91,2] = PR[GP1:90,2] + 15.790;
   1:L PR[91] 10mm/sec CNT100;
   1:  PR[GP1:91,1] = PR[GP1:90,1] + -24.446;
   1:  PR[GP1:91,2] = PR[GP1:90,2] + 15.475;
   1:L PR[91] 10mm/sec CNT100;
   1:  PR[GP1:91,1] = PR[GP1:90,1] + -26.740;
   1:  PR[GP1:91,2] = PR[GP1:90,2] + 14.502;
   1:L PR[91] 10mm/sec CNT100;
   1:  PR[GP1:91,1] = PR[GP1:90,1] + -27.616;
   1:  PR[GP1:91,2] = PR[GP1:90,2] + 14.069;
   1:L PR[91] 10mm/sec CNT100;
   1:  PR[GP1:91,1] = PR[GP1:90,1] + -29.833;
   1:  PR[GP1:91,2] = PR[GP1:90,2] + 12.512;
   1:L PR[91] 10mm/sec CNT100;
   1:  PR[GP1:91,1] = PR[GP1:90,1] + -30.453;
   1:  PR[GP1:91,2] = PR[GP1:90,2] + 12.031;
   1:L PR[91] 10mm/sec CNT100;
   1:  PR[GP1:91,1] = PR[GP1:90,1] + -32.389;
   1:  PR[GP1:91,2] = PR[GP1:90,2] + 9.933;
   1:L PR[91] 10mm/sec CNT100;
   1:  PR[GP1:91,1] = PR[GP1:90,1] + -32.814;
   1:  PR[GP1:91,2] = PR[GP1:90,2] + 9.436;
   1:L PR[91] 10mm/sec CNT100;
   1:  PR[GP1:91,1] = PR[GP1:90,1] + -34.303;
   1:  PR[GP1:91,2] = PR[GP1:90,2] + 6.904;
   1:L PR[91] 10mm/sec CNT100;
   1:  PR[GP1:91,1] = PR[GP1:90,1] + -34.585;
   1:  PR[GP1:91,2] = PR[GP1:90,2] + 6.394;
   1:L PR[91] 10mm/sec CNT100;
   1:  PR[GP1:91,1] = PR[GP1:90,1] + -35.683;
   1:  PR[GP1:91,2] = PR[GP1:90,2] + 3.038;
   1:L PR[91] 10mm/sec CNT100;
   1:  PR[GP1:91,1] = PR[GP1:90,1] + -35.982;
   1:  PR[GP1:91,2] = PR[GP1:90,2] + 0.110;
   1:L PR[91] 10mm/sec CNT100;
   1:  PR[GP1:91,1] = PR[GP1:90,1] + -36.077;
   1:  PR[GP1:91,2] = PR[GP1:90,2] + -0.479;
   1:L PR[91] 10mm/sec CNT100;
   1:  PR[GP1:91,1] = PR[GP1:90,1] + -35.863;
   1:  PR[GP1:91,2] = PR[GP1:90,2] + -2.406;
   1:L PR[91] 10mm/sec CNT100;
   1:  PR[GP1:91,1] = PR[GP1:90,1] + -35.719;
   1:  PR[GP1:91,2] = PR[GP1:90,2] + -3.281;
   1:L PR[91] 10mm/sec CNT100;
   1:  PR[GP1:91,1] = PR[GP1:90,1] + -35.639;
   1:  PR[GP1:91,2] = PR[GP1:90,2] + -3.991;
   1:L PR[91] 10mm/sec CNT100;
   1:  PR[GP1:91,1] = PR[GP1:90,1] + -35.403;
   1:  PR[GP1:91,2] = PR[GP1:90,2] + -4.735;
   1:L PR[91] 10mm/sec CNT100;
   1:  PR[GP1:91,1] = PR[GP1:90,1] + -34.530;
   1:  PR[GP1:91,2] = PR[GP1:90,2] + -7.335;
   1:L PR[91] 10mm/sec CNT100;
   1:  PR[GP1:91,1] = PR[GP1:90,1] + -34.050;
   1:  PR[GP1:91,2] = PR[GP1:90,2] + -8.188;
   1:L PR[91] 10mm/sec CNT100;
   1:  PR[GP1:91,1] = PR[GP1:90,1] + -32.752;
   1:  PR[GP1:91,2] = PR[GP1:90,2] + -10.369;
   1:L PR[91] 10mm/sec CNT100;
   1:  PR[GP1:91,1] = PR[GP1:90,1] + -31.935;
   1:  PR[GP1:91,2] = PR[GP1:90,2] + -11.310;
   1:L PR[91] 10mm/sec CNT100;
   1:  PR[GP1:91,1] = PR[GP1:90,1] + -30.406;
   1:  PR[GP1:91,2] = PR[GP1:90,2] + -12.960;
   1:L PR[91] 10mm/sec CNT100;
   1:  PR[GP1:91,1] = PR[GP1:90,1] + -29.149;
   1:  PR[GP1:91,2] = PR[GP1:90,2] + -13.927;
   1:L PR[91] 10mm/sec CNT100;
   1:  PR[GP1:91,1] = PR[GP1:90,1] + -27.620;
   1:  PR[GP1:91,2] = PR[GP1:90,2] + -15.005;
   1:L PR[91] 10mm/sec CNT100;
   1:  PR[GP1:91,1] = PR[GP1:90,1] + -25.820;
   1:  PR[GP1:91,2] = PR[GP1:90,2] + -15.888;
   1:L PR[91] 10mm/sec CNT100;
   1:  PR[GP1:91,1] = PR[GP1:90,1] + -24.532;
   1:  PR[GP1:91,2] = PR[GP1:90,2] + -16.441;
   1:L PR[91] 10mm/sec CNT100;
   1:  PR[GP1:91,1] = PR[GP1:90,1] + -21.344;
   1:  PR[GP1:91,2] = PR[GP1:90,2] + -17.273;
   1:  PR[GP1:91,3] = PR[GP1:90,3] + 14.300;
   1:L PR[91] 10mm/sec CNT100;
   1:  PR[GP1:91,1] = PR[GP1:90,1] + -18.214;
   1:  PR[GP1:91,2] = PR[GP1:90,2] + -17.492;
   1:L PR[91] 10mm/sec CNT100;
   1:  PR[GP1:91,1] = PR[GP1:90,1] + -17.711;
   1:  PR[GP1:91,2] = PR[GP1:90,2] + -17.511;
   1:L PR[91] 10mm/sec CNT100;
   1:  PR[GP1:91,1] = PR[GP1:90,1] + -15.208;
   1:  PR[GP1:91,2] = PR[GP1:90,2] + -17.199;
   1:L PR[91] 10mm/sec CNT100;
   1:  PR[GP1:91,1] = PR[GP1:90,1] + -14.060;
   1:  PR[GP1:91,2] = PR[GP1:90,2] + -17.013;
   1:L PR[91] 10mm/sec CNT100;
   1:  PR[GP1:91,1] = PR[GP1:90,1] + -12.333;
   1:  PR[GP1:91,2] = PR[GP1:90,2] + -16.438;
   1:L PR[91] 10mm/sec CNT100;
   1:  PR[GP1:91,1] = PR[GP1:90,1] + -10.584;
   1:  PR[GP1:91,2] = PR[GP1:90,2] + -15.777;
   1:L PR[91] 10mm/sec CNT100;
   1:  PR[GP1:91,1] = PR[GP1:90,1] + -9.640;
   1:  PR[GP1:91,2] = PR[GP1:90,2] + -15.234;
   1:L PR[91] 10mm/sec CNT100;
   1:  PR[GP1:91,1] = PR[GP1:90,1] + -7.456;
   1:  PR[GP1:91,2] = PR[GP1:90,2] + -13.845;
   1:L PR[91] 10mm/sec CNT100;
   1:  PR[GP1:91,1] = PR[GP1:90,1] + -7.174;
   1:  PR[GP1:91,2] = PR[GP1:90,2] + -13.593;
   1:L PR[91] 10mm/sec CNT100;
   1:  PR[GP1:91,1] = PR[GP1:90,1] + -5.487;
   1:  PR[GP1:91,2] = PR[GP1:90,2] + -11.937;
   1:L PR[91] 10mm/sec CNT100;
   1:  PR[GP1:91,1] = PR[GP1:90,1] + -4.898;
   1:  PR[GP1:91,2] = PR[GP1:90,2] + -11.390;
   1:L PR[91] 10mm/sec CNT100;
   1:  PR[GP1:91,1] = PR[GP1:90,1] + -4.828;
   1:  PR[GP1:91,2] = PR[GP1:90,2] + -11.312;
   1:L PR[91] 10mm/sec CNT100;
   1:  PR[GP1:91,1] = PR[GP1:90,1] + -2.822;
   1:  PR[GP1:91,2] = PR[GP1:90,2] + -8.356;
   1:L PR[91] 10mm/sec CNT100;
   1:  PR[GP1:91,1] = PR[GP1:90,1] + -2.321;
   1:  PR[GP1:91,2] = PR[GP1:90,2] + -7.835;
   1:L PR[91] 10mm/sec CNT100;
   1:  PR[GP1:91,1] = PR[GP1:90,1] + -1.828;
   1:  PR[GP1:91,2] = PR[GP1:90,2] + -7.505;
   1:L PR[91] 10mm/sec CNT100;
   1:  PR[GP1:91,1] = PR[GP1:90,1] + -1.236;
   1:  PR[GP1:91,2] = PR[GP1:90,2] + -7.328;
   1:L PR[91] 10mm/sec CNT100;
   1:  PR[GP1:91,1] = PR[GP1:90,1] + -0.616;
   1:  PR[GP1:91,2] = PR[GP1:90,2] + -7.288;
   1:L PR[91] 10mm/sec CNT100;
   1:  PR[GP1:91,1] = PR[GP1:90,1] + -0.026;
   1:  PR[GP1:91,2] = PR[GP1:90,2] + -7.473;
   1:L PR[91] 10mm/sec CNT100;
   1:  PR[GP1:91,1] = PR[GP1:90,1] + 0.504;
   1:  PR[GP1:91,2] = PR[GP1:90,2] + -7.755;
   1:L PR[91] 10mm/sec CNT100;
   1:  PR[GP1:91,1] = PR[GP1:90,1] + 1.029;
   1:  PR[GP1:91,2] = PR[GP1:90,2] + -8.333;
   1:L PR[91] 10mm/sec CNT100;
   1:  PR[GP1:91,1] = PR[GP1:90,1] + 1.143;
   1:  PR[GP1:91,2] = PR[GP1:90,2] + -8.591;
   1:L PR[91] 10mm/sec CNT100;
   1:  PR[GP1:91,1] = PR[GP1:90,1] + 1.486;
   1:  PR[GP1:91,2] = PR[GP1:90,2] + -9.203;
   1:L PR[91] 10mm/sec CNT100;
   1:  PR[GP1:91,1] = PR[GP1:90,1] + 1.708;
   1:  PR[GP1:91,2] = PR[GP1:90,2] + -9.563;
   1:L PR[91] 10mm/sec CNT100;
   1:  PR[GP1:91,1] = PR[GP1:90,1] + 2.858;
   1:  PR[GP1:91,2] = PR[GP1:90,2] + -11.121;
   1:L PR[91] 10mm/sec CNT100;
   1:  PR[GP1:91,1] = PR[GP1:90,1] + 3.489;
   1:  PR[GP1:91,2] = PR[GP1:90,2] + -11.878;
   1:L PR[91] 10mm/sec CNT100;
   1:  PR[GP1:91,1] = PR[GP1:90,1] + 4.902;
   1:  PR[GP1:91,2] = PR[GP1:90,2] + -13.225;
   1:L PR[91] 10mm/sec CNT100;
   1:  PR[GP1:91,1] = PR[GP1:90,1] + 5.373;
   1:  PR[GP1:91,2] = PR[GP1:90,2] + -13.634;
   1:L PR[91] 10mm/sec CNT100;
   1:  PR[GP1:91,1] = PR[GP1:90,1] + 7.538;
   1:  PR[GP1:91,2] = PR[GP1:90,2] + -15.106;
   1:L PR[91] 10mm/sec CNT100;
   1:  PR[GP1:91,1] = PR[GP1:90,1] + 9.935;
   1:  PR[GP1:91,2] = PR[GP1:90,2] + -16.266;
   1:L PR[91] 10mm/sec CNT100;
   1:  PR[GP1:91,1] = PR[GP1:90,1] + 10.674;
   1:  PR[GP1:91,2] = PR[GP1:90,2] + -16.515;
   1:L PR[91] 10mm/sec CNT100;
   1:  PR[GP1:91,1] = PR[GP1:90,1] + 12.508;
   1:  PR[GP1:91,2] = PR[GP1:90,2] + -17.087;
   1:L PR[91] 10mm/sec CNT100;
   1:  PR[GP1:91,1] = PR[GP1:90,1] + 14.542;
   1:  PR[GP1:91,2] = PR[GP1:90,2] + -17.446;
   1:L PR[91] 10mm/sec CNT100;
   1:  PR[GP1:91,1] = PR[GP1:90,1] + 15.216;
   1:  PR[GP1:91,2] = PR[GP1:90,2] + -17.551;
   1:L PR[91] 10mm/sec CNT100;
   1:  PR[GP1:91,1] = PR[GP1:90,1] + 18.061;
   1:  PR[GP1:91,2] = PR[GP1:90,2] + -17.648;
   1:L PR[91] 10mm/sec CNT100;
   1:  PR[GP1:91,1] = PR[GP1:90,1] + 20.946;
   1:  PR[GP1:91,2] = PR[GP1:90,2] + -17.342;
   1:L PR[91] 10mm/sec CNT100;
   1:  PR[GP1:91,1] = PR[GP1:90,1] + 23.739;
   1:  PR[GP1:91,2] = PR[GP1:90,2] + -16.625;
   1:L PR[91] 10mm/sec CNT100;
   1:  PR[GP1:91,1] = PR[GP1:90,1] + 26.317;
   1:  PR[GP1:91,2] = PR[GP1:90,2] + -15.538;
   1:L PR[91] 10mm/sec CNT100;
   1:  PR[GP1:91,1] = PR[GP1:90,1] + 28.665;
   1:  PR[GP1:91,2] = PR[GP1:90,2] + -14.098;
   1:L PR[91] 10mm/sec CNT100;
   1:  PR[GP1:91,1] = PR[GP1:90,1] + 30.753;
   1:  PR[GP1:91,2] = PR[GP1:90,2] + -12.334;
   1:L PR[91] 10mm/sec CNT100;
   1:  PR[GP1:91,1] = PR[GP1:90,1] + 32.532;
   1:  PR[GP1:91,2] = PR[GP1:90,2] + -10.289;
   1:L PR[91] 10mm/sec CNT100;
   1:  PR[GP1:91,1] = PR[GP1:90,1] + 33.960;
   1:  PR[GP1:91,2] = PR[GP1:90,2] + -8.013;
   1:L PR[91] 10mm/sec CNT100;
   1:  PR[GP1:91,1] = PR[GP1:90,1] + 35.006;
   1:  PR[GP1:91,2] = PR[GP1:90,2] + -5.563;
   1:L PR[91] 10mm/sec CNT100;
   1:  PR[GP1:91,1] = PR[GP1:90,1] + 35.628;
   1:  PR[GP1:91,2] = PR[GP1:90,2] + -2.996;
   1:L PR[91] 10mm/sec CNT100;
   1:  PR[GP1:91,1] = PR[GP1:90,1] + 35.840;
   1:  PR[GP1:91,2] = PR[GP1:90,2] + -0.375;
   1:L PR[91] 10mm/sec CNT100;
   1:  PR[GP1:91,1] = PR[GP1:90,1] + 35.491;
   1:  PR[GP1:91,2] = PR[GP1:90,2] + 2.944;
   1:L PR[91] 10mm/sec CNT100;
   1:  PR[GP1:91,1] = PR[GP1:90,1] + 34.487;
   1:  PR[GP1:91,2] = PR[GP1:90,2] + 6.126;
   1:L PR[91] 10mm/sec CNT100;
   1:  PR[GP1:91,1] = PR[GP1:90,1] + 32.847;
   1:  PR[GP1:91,2] = PR[GP1:90,2] + 9.049;
   1:L PR[91] 10mm/sec CNT100;
   1:  PR[GP1:91,1] = PR[GP1:90,1] + 30.637;
   1:  PR[GP1:91,2] = PR[GP1:90,2] + 11.603;
   1:L PR[91] 10mm/sec CNT100;
   1:  PR[GP1:91,1] = PR[GP1:90,1] + 27.942;
   1:  PR[GP1:91,2] = PR[GP1:90,2] + 13.686;
   1:L PR[91] 10mm/sec CNT100;
   1:  PR[GP1:91,1] = PR[GP1:90,1] + 24.870;
   1:  PR[GP1:91,2] = PR[GP1:90,2] + 15.217;
   1:L PR[91] 10mm/sec CNT100;
   1:  PR[GP1:91,1] = PR[GP1:90,1] + 21.522;
   1:  PR[GP1:91,2] = PR[GP1:90,2] + 16.132;
   1:L PR[91] 10mm/sec CNT100;
   1:  PR[GP1:91,1] = PR[GP1:90,1] + 17.966;
   1:  PR[GP1:91,2] = PR[GP1:90,2] + 16.388;
   1:L PR[91] 10mm/sec CNT100;
   1:  PR[GP1:91,1] = PR[GP1:90,1] + 14.409;
   1:  PR[GP1:91,2] = PR[GP1:90,2] + 15.984;
   1:L PR[91] 10mm/sec CNT100;
   1:  PR[GP1:91,1] = PR[GP1:90,1] + 10.912;
   1:  PR[GP1:91,2] = PR[GP1:90,2] + 14.914;
   1:L PR[91] 10mm/sec CNT100;
   1:  PR[GP1:91,1] = PR[GP1:90,1] + 7.689;
   1:  PR[GP1:91,2] = PR[GP1:90,2] + 13.240;
   1:L PR[91] 10mm/sec CNT100;
   1:  PR[GP1:91,1] = PR[GP1:90,1] + 4.842;
   1:  PR[GP1:91,2] = PR[GP1:90,2] + 11.020;
   1:L PR[91] 10mm/sec CNT100;
   1:  PR[GP1:91,1] = PR[GP1:90,1] + 2.497;
   1:  PR[GP1:91,2] = PR[GP1:90,2] + 8.329;
   1:L PR[91] 10mm/sec CNT100;
   1:  PR[GP1:91,1] = PR[GP1:90,1] + 2.331;
   1:  PR[GP1:91,2] = PR[GP1:90,2] + 8.087;
   1:L PR[91] 10mm/sec CNT100;
   1:  PR[GP1:91,1] = PR[GP1:90,1] + 1.364;
   1:  PR[GP1:91,2] = PR[GP1:90,2] + 6.440;
   1:L PR[91] 10mm/sec CNT100;
   1:  PR[GP1:91,1] = PR[GP1:90,1] + 1.030;
   1:  PR[GP1:91,2] = PR[GP1:90,2] + 6.079;
   1:L PR[91] 10mm/sec CNT100;
   1:  PR[GP1:91,1] = PR[GP1:90,1] + 0.533;
   1:  PR[GP1:91,2] = PR[GP1:90,2] + 5.481;
   1:L PR[91] 10mm/sec CNT100;
   1:  PR[GP1:91,1] = PR[GP1:90,1] + -0.297;
   1:  PR[GP1:91,2] = PR[GP1:90,2] + 5.198;
   1:L PR[91] 10mm/sec CNT100;
   1:  PR[GP1:91,1] = PR[GP1:90,1] + -0.857;
   1:  PR[GP1:91,2] = PR[GP1:90,2] + 5.079;
   1:L PR[91] 10mm/sec CNT100;
   1:  PR[GP1:91,1] = PR[GP1:90,1] + -1.475;
   1:  PR[GP1:91,2] = PR[GP1:90,2] + 5.343;
   1:L PR[91] 10mm/sec CNT100;
   1:  PR[GP1:91,1] = PR[GP1:90,1] + -2.116;
   1:  PR[GP1:91,2] = PR[GP1:90,2] + 5.483;
   1:L PR[91] 10mm/sec CNT100;
   1:  PR[GP1:91,1] = PR[GP1:90,1] + -2.866;
   1:  PR[GP1:91,2] = PR[GP1:90,2] + 6.360;
   1:L PR[91] 10mm/sec CNT100;
   1:  PR[GP1:91,1] = PR[GP1:90,1] + -3.054;
   1:  PR[GP1:91,2] = PR[GP1:90,2] + 6.543;
   1:L PR[91] 10mm/sec CNT100;
   1:  PR[GP1:91,1] = PR[GP1:90,1] + -3.589;
   1:  PR[GP1:91,2] = PR[GP1:90,2] + 7.593;
   1:L PR[91] 10mm/sec CNT100;
   1:  PR[GP1:91,1] = PR[GP1:90,1] + -4.664;
   1:  PR[GP1:91,2] = PR[GP1:90,2] + 9.053;
   1:L PR[91] 10mm/sec CNT100;
   1:  PR[GP1:91,1] = PR[GP1:90,1] + -5.767;
   1:  PR[GP1:91,2] = PR[GP1:90,2] + 10.478;
   1:L PR[91] 10mm/sec CNT100;
   1:  PR[GP1:91,1] = PR[GP1:90,1] + -6.598;
   1:  PR[GP1:91,2] = PR[GP1:90,2] + 11.234;
   1:L PR[91] 10mm/sec CNT100;
   1:  PR[GP1:91,1] = PR[GP1:90,1] + -8.472;
   1:  PR[GP1:91,2] = PR[GP1:90,2] + 12.866;
   1:L PR[91] 10mm/sec CNT100;
   1:  PR[GP1:91,1] = PR[GP1:90,1] + -11.571;
   1:  PR[GP1:91,2] = PR[GP1:90,2] + 14.666;
   1:L PR[91] 10mm/sec CNT100;
   1:  PR[GP1:91,1] = PR[GP1:90,1] + -14.592;
   1:  PR[GP1:91,2] = PR[GP1:90,2] + 15.731;
   1:L PR[91] 10mm/sec CNT100;
   1:  PR[GP1:91,1] = PR[GP1:90,1] + -15.151;
   1:  PR[GP1:91,2] = PR[GP1:90,2] + 15.860;
   1:L PR[91] 10mm/sec CNT100;
   1:  PR[GP1:91,1] = PR[GP1:90,1] + -17.809;
   1:  PR[GP1:91,2] = PR[GP1:90,2] + 16.234;
   1:L PR[91] 10mm/sec CNT100;
   1:  PR[GP1:91,1] = PR[GP1:90,1] + -18.897;
   1:  PR[GP1:91,2] = PR[GP1:90,2] + 16.254;
   1:L PR[91] 10mm/sec CNT100;
   1:  PR[GP1:91,1] = PR[GP1:90,1] + -21.138;
   1:  PR[GP1:91,2] = PR[GP1:90,2] + 16.122;
   1:L PR[91] 10mm/sec CNT100;
   1:  PR[GP1:91,1] = PR[GP1:90,1] + -22.620;
   1:  PR[GP1:91,2] = PR[GP1:90,2] + 15.835;
   1:L PR[91] 10mm/sec CNT100;
   1:  PR[GP1:91,1] = PR[GP1:90,1] + -24.437;
   1:  PR[GP1:91,2] = PR[GP1:90,2] + 15.355;
   1:L PR[91] 10mm/sec CNT100;
   1:  PR[GP1:91,1] = PR[GP1:90,1] + -26.133;
   1:  PR[GP1:91,2] = PR[GP1:90,2] + 14.636;
   1:L PR[91] 10mm/sec CNT100;
   1:  PR[GP1:91,1] = PR[GP1:90,1] + -27.557;
   1:  PR[GP1:91,2] = PR[GP1:90,2] + 13.933;
   1:L PR[91] 10mm/sec CNT100;
   1:  PR[GP1:91,1] = PR[GP1:90,1] + -29.268;
   1:  PR[GP1:91,2] = PR[GP1:90,2] + 12.730;
   1:L PR[91] 10mm/sec CNT100;
   1:  PR[GP1:91,1] = PR[GP1:90,1] + -30.349;
   1:  PR[GP1:91,2] = PR[GP1:90,2] + 11.891;
   1:L PR[91] 10mm/sec CNT100;
   1:  PR[GP1:91,1] = PR[GP1:90,1] + -31.884;
   1:  PR[GP1:91,2] = PR[GP1:90,2] + 10.229;
   1:L PR[91] 10mm/sec CNT100;
   1:  PR[GP1:91,1] = PR[GP1:90,1] + -32.673;
   1:  PR[GP1:91,2] = PR[GP1:90,2] + 9.304;
   1:L PR[91] 10mm/sec CNT100;
   1:  PR[GP1:91,1] = PR[GP1:90,1] + -33.871;
   1:  PR[GP1:91,2] = PR[GP1:90,2] + 7.267;
   1:L PR[91] 10mm/sec CNT100;
   1:  PR[GP1:91,1] = PR[GP1:90,1] + -34.416;
   1:  PR[GP1:91,2] = PR[GP1:90,2] + 6.279;
   1:L PR[91] 10mm/sec CNT100;
   1:  PR[GP1:91,1] = PR[GP1:90,1] + -35.169;
   1:  PR[GP1:91,2] = PR[GP1:90,2] + 3.999;
   1:L PR[91] 10mm/sec CNT100;
   1:  PR[GP1:91,1] = PR[GP1:90,1] + -35.498;
   1:  PR[GP1:91,2] = PR[GP1:90,2] + 2.951;
   1:L PR[91] 10mm/sec CNT100;
   1:  PR[GP1:91,1] = PR[GP1:90,1] + -35.741;
   1:  PR[GP1:91,2] = PR[GP1:90,2] + 0.572;
   1:L PR[91] 10mm/sec CNT100;
   1:  PR[GP1:91,1] = PR[GP1:90,1] + -35.920;
   1:  PR[GP1:91,2] = PR[GP1:90,2] + -0.530;
   1:L PR[91] 10mm/sec CNT100;
   1:  PR[GP1:91,1] = PR[GP1:90,1] + -35.834;
   1:  PR[GP1:91,2] = PR[GP1:90,2] + -1.305;
   1:L PR[91] 10mm/sec CNT100;
   1:  PR[GP1:91,1] = PR[GP1:90,1] + -35.589;
   1:  PR[GP1:91,2] = PR[GP1:90,2] + -2.790;
   1:L PR[91] 10mm/sec CNT100;
   1:  PR[GP1:91,1] = PR[GP1:90,1] + -35.451;
   1:  PR[GP1:91,2] = PR[GP1:90,2] + -4.028;
   1:L PR[91] 10mm/sec CNT100;
   1:  PR[GP1:91,1] = PR[GP1:90,1] + -35.035;
   1:  PR[GP1:91,2] = PR[GP1:90,2] + -5.337;
   1:L PR[91] 10mm/sec CNT100;
   1:  PR[GP1:91,1] = PR[GP1:90,1] + -34.361;
   1:  PR[GP1:91,2] = PR[GP1:90,2] + -7.346;
   1:L PR[91] 10mm/sec CNT100;
   1:  PR[GP1:91,1] = PR[GP1:90,1] + -33.573;
   1:  PR[GP1:91,2] = PR[GP1:90,2] + -8.744;
   1:L PR[91] 10mm/sec CNT100;
   1:  PR[GP1:91,1] = PR[GP1:90,1] + -32.612;
   1:  PR[GP1:91,2] = PR[GP1:90,2] + -10.359;
   1:L PR[91] 10mm/sec CNT100;
   1:  PR[GP1:91,1] = PR[GP1:90,1] + -31.358;
   1:  PR[GP1:91,2] = PR[GP1:90,2] + -11.803;
   1:L PR[91] 10mm/sec CNT100;
   1:  PR[GP1:91,1] = PR[GP1:90,1] + -30.307;
   1:  PR[GP1:91,2] = PR[GP1:90,2] + -12.937;
   1:L PR[91] 10mm/sec CNT100;
   1:  PR[GP1:91,1] = PR[GP1:90,1] + -28.486;
   1:  PR[GP1:91,2] = PR[GP1:90,2] + -14.339;
   1:L PR[91] 10mm/sec CNT100;
   1:  PR[GP1:91,1] = PR[GP1:90,1] + -27.572;
   1:  PR[GP1:91,2] = PR[GP1:90,2] + -14.983;
   1:L PR[91] 10mm/sec CNT100;
   1:  PR[GP1:91,1] = PR[GP1:90,1] + -25.087;
   1:  PR[GP1:91,2] = PR[GP1:90,2] + -16.202;
   1:L PR[91] 10mm/sec CNT100;
   1:  PR[GP1:91,1] = PR[GP1:90,1] + -24.545;
   1:  PR[GP1:91,2] = PR[GP1:90,2] + -16.434;
   1:L PR[91] 10mm/sec CNT100;
   1:  PR[GP1:91,1] = PR[GP1:90,1] + -21.546;
   1:  PR[GP1:91,2] = PR[GP1:90,2] + -17.246;
   1:  PR[GP1:91,3] = PR[GP1:90,3] + 15.400;
   1:L PR[91] 10mm/sec CNT100;
   1:  PR[GP1:91,1] = PR[GP1:90,1] + -20.923;
   1:  PR[GP1:91,2] = PR[GP1:90,2] + -17.395;
   1:L PR[91] 10mm/sec CNT100;
   1:  PR[GP1:91,1] = PR[GP1:90,1] + -18.530;
   1:  PR[GP1:91,2] = PR[GP1:90,2] + -17.564;
   1:L PR[91] 10mm/sec CNT100;
   1:  PR[GP1:91,1] = PR[GP1:90,1] + -17.233;
   1:  PR[GP1:91,2] = PR[GP1:90,2] + -17.615;
   1:L PR[91] 10mm/sec CNT100;
   1:  PR[GP1:91,1] = PR[GP1:90,1] + -15.559;
   1:  PR[GP1:91,2] = PR[GP1:90,2] + -17.406;
   1:L PR[91] 10mm/sec CNT100;
   1:  PR[GP1:91,1] = PR[GP1:90,1] + -13.553;
   1:  PR[GP1:91,2] = PR[GP1:90,2] + -17.082;
   1:L PR[91] 10mm/sec CNT100;
   1:  PR[GP1:91,1] = PR[GP1:90,1] + -12.695;
   1:  PR[GP1:91,2] = PR[GP1:90,2] + -16.796;
   1:L PR[91] 10mm/sec CNT100;
   1:  PR[GP1:91,1] = PR[GP1:90,1] + -10.066;
   1:  PR[GP1:91,2] = PR[GP1:90,2] + -15.801;
   1:L PR[91] 10mm/sec CNT100;
   1:  PR[GP1:91,1] = PR[GP1:90,1] + -9.458;
   1:  PR[GP1:91,2] = PR[GP1:90,2] + -15.422;
   1:L PR[91] 10mm/sec CNT100;
   1:  PR[GP1:91,1] = PR[GP1:90,1] + -7.270;
   1:  PR[GP1:91,2] = PR[GP1:90,2] + -14.127;
   1:L PR[91] 10mm/sec CNT100;
   1:  PR[GP1:91,1] = PR[GP1:90,1] + -6.756;
   1:  PR[GP1:91,2] = PR[GP1:90,2] + -13.767;
   1:L PR[91] 10mm/sec CNT100;
   1:  PR[GP1:91,1] = PR[GP1:90,1] + -4.949;
   1:  PR[GP1:91,2] = PR[GP1:90,2] + -12.088;
   1:L PR[91] 10mm/sec CNT100;
   1:  PR[GP1:91,1] = PR[GP1:90,1] + -4.007;
   1:  PR[GP1:91,2] = PR[GP1:90,2] + -11.042;
   1:L PR[91] 10mm/sec CNT100;
   1:  PR[GP1:91,1] = PR[GP1:90,1] + -2.976;
   1:  PR[GP1:91,2] = PR[GP1:90,2] + -9.519;
   1:L PR[91] 10mm/sec CNT100;
   1:  PR[GP1:91,1] = PR[GP1:90,1] + -2.253;
   1:  PR[GP1:91,2] = PR[GP1:90,2] + -8.769;
   1:L PR[91] 10mm/sec CNT100;
   1:  PR[GP1:91,1] = PR[GP1:90,1] + -1.990;
   1:  PR[GP1:91,2] = PR[GP1:90,2] + -8.593;
   1:L PR[91] 10mm/sec CNT100;
   1:  PR[GP1:91,1] = PR[GP1:90,1] + -1.131;
   1:  PR[GP1:91,2] = PR[GP1:90,2] + -8.336;
   1:L PR[91] 10mm/sec CNT100;
   1:  PR[GP1:91,1] = PR[GP1:90,1] + -0.769;
   1:  PR[GP1:91,2] = PR[GP1:90,2] + -8.313;
   1:L PR[91] 10mm/sec CNT100;
   1:  PR[GP1:91,1] = PR[GP1:90,1] + 0.090;
   1:  PR[GP1:91,2] = PR[GP1:90,2] + -8.582;
   1:L PR[91] 10mm/sec CNT100;
   1:  PR[GP1:91,1] = PR[GP1:90,1] + 0.375;
   1:  PR[GP1:91,2] = PR[GP1:90,2] + -8.733;
   1:L PR[91] 10mm/sec CNT100;
   1:  PR[GP1:91,1] = PR[GP1:90,1] + 1.101;
   1:  PR[GP1:91,2] = PR[GP1:90,2] + -9.532;
   1:L PR[91] 10mm/sec CNT100;
   1:  PR[GP1:91,1] = PR[GP1:90,1] + 1.233;
   1:  PR[GP1:91,2] = PR[GP1:90,2] + -9.769;
   1:L PR[91] 10mm/sec CNT100;
   1:  PR[GP1:91,1] = PR[GP1:90,1] + 2.036;
   1:  PR[GP1:91,2] = PR[GP1:90,2] + -10.875;
   1:L PR[91] 10mm/sec CNT100;
   1:  PR[GP1:91,1] = PR[GP1:90,1] + 3.145;
   1:  PR[GP1:91,2] = PR[GP1:90,2] + -12.205;
   1:L PR[91] 10mm/sec CNT100;
   1:  PR[GP1:91,1] = PR[GP1:90,1] + 3.981;
   1:  PR[GP1:91,2] = PR[GP1:90,2] + -13.002;
   1:L PR[91] 10mm/sec CNT100;
   1:  PR[GP1:91,1] = PR[GP1:90,1] + 5.052;
   1:  PR[GP1:91,2] = PR[GP1:90,2] + -13.931;
   1:L PR[91] 10mm/sec CNT100;
   1:  PR[GP1:91,1] = PR[GP1:90,1] + 6.410;
   1:  PR[GP1:91,2] = PR[GP1:90,2] + -14.859;
   1:L PR[91] 10mm/sec CNT100;
   1:  PR[GP1:91,1] = PR[GP1:90,1] + 7.217;
   1:  PR[GP1:91,2] = PR[GP1:90,2] + -15.363;
   1:L PR[91] 10mm/sec CNT100;
   1:  PR[GP1:91,1] = PR[GP1:90,1] + 9.317;
   1:  PR[GP1:91,2] = PR[GP1:90,2] + -16.355;
   1:L PR[91] 10mm/sec CNT100;
   1:  PR[GP1:91,1] = PR[GP1:90,1] + 9.601;
   1:  PR[GP1:91,2] = PR[GP1:90,2] + -16.477;
   1:L PR[91] 10mm/sec CNT100;
   1:  PR[GP1:91,1] = PR[GP1:90,1] + 12.187;
   1:  PR[GP1:91,2] = PR[GP1:90,2] + -17.267;
   1:L PR[91] 10mm/sec CNT100;
   1:  PR[GP1:91,1] = PR[GP1:90,1] + 12.839;
   1:  PR[GP1:91,2] = PR[GP1:90,2] + -17.381;
   1:L PR[91] 10mm/sec CNT100;
   1:  PR[GP1:91,1] = PR[GP1:90,1] + 14.890;
   1:  PR[GP1:91,2] = PR[GP1:90,2] + -17.702;
   1:L PR[91] 10mm/sec CNT100;
   1:  PR[GP1:91,1] = PR[GP1:90,1] + 17.675;
   1:  PR[GP1:91,2] = PR[GP1:90,2] + -17.767;
   1:L PR[91] 10mm/sec CNT100;
   1:  PR[GP1:91,1] = PR[GP1:90,1] + 20.516;
   1:  PR[GP1:91,2] = PR[GP1:90,2] + -17.450;
   1:L PR[91] 10mm/sec CNT100;
   1:  PR[GP1:91,1] = PR[GP1:90,1] + 23.320;
   1:  PR[GP1:91,2] = PR[GP1:90,2] + -16.728;
   1:L PR[91] 10mm/sec CNT100;
   1:  PR[GP1:91,1] = PR[GP1:90,1] + 25.967;
   1:  PR[GP1:91,2] = PR[GP1:90,2] + -15.617;
   1:L PR[91] 10mm/sec CNT100;
   1:  PR[GP1:91,1] = PR[GP1:90,1] + 27.186;
   1:  PR[GP1:91,2] = PR[GP1:90,2] + -14.879;
   1:L PR[91] 10mm/sec CNT100;
   1:  PR[GP1:91,1] = PR[GP1:90,1] + 28.355;
   1:  PR[GP1:91,2] = PR[GP1:90,2] + -14.161;
   1:L PR[91] 10mm/sec CNT100;
   1:  PR[GP1:91,1] = PR[GP1:90,1] + 30.444;
   1:  PR[GP1:91,2] = PR[GP1:90,2] + -12.392;
   1:L PR[91] 10mm/sec CNT100;
   1:  PR[GP1:91,1] = PR[GP1:90,1] + 32.223;
   1:  PR[GP1:91,2] = PR[GP1:90,2] + -10.341;
   1:L PR[91] 10mm/sec CNT100;
   1:  PR[GP1:91,1] = PR[GP1:90,1] + 33.651;
   1:  PR[GP1:91,2] = PR[GP1:90,2] + -8.060;
   1:L PR[91] 10mm/sec CNT100;
   1:  PR[GP1:91,1] = PR[GP1:90,1] + 34.696;
   1:  PR[GP1:91,2] = PR[GP1:90,2] + -5.603;
   1:L PR[91] 10mm/sec CNT100;
   1:  PR[GP1:91,1] = PR[GP1:90,1] + 35.334;
   1:  PR[GP1:91,2] = PR[GP1:90,2] + -3.028;
   1:L PR[91] 10mm/sec CNT100;
   1:  PR[GP1:91,1] = PR[GP1:90,1] + 35.514;
